RoboDK station: kr30 cnc 041619 kinda works.rdk

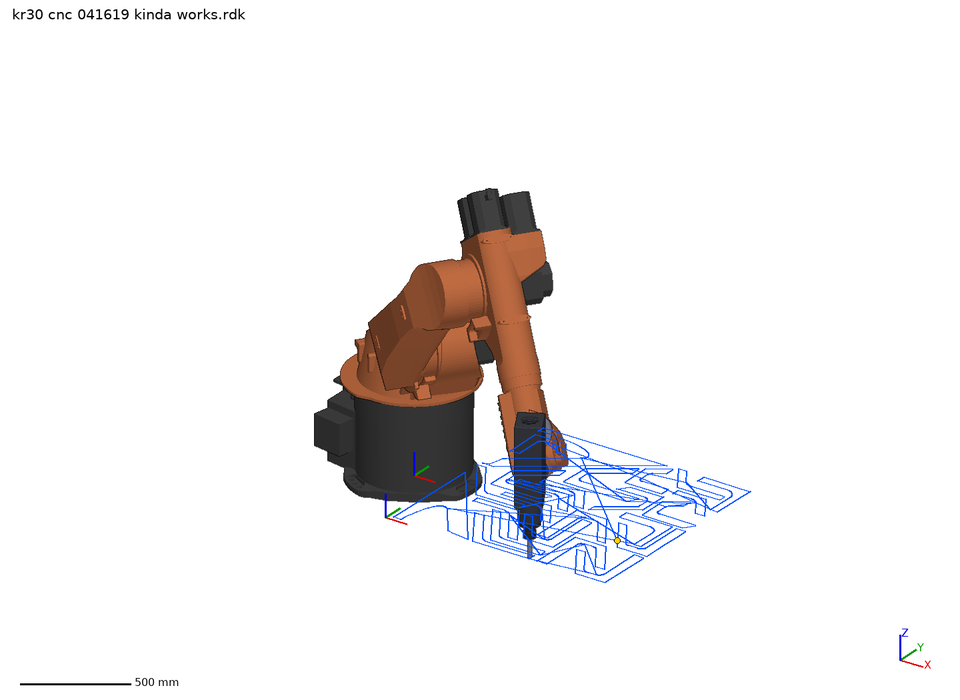
[picture v0: the station drawn from its stored meshes, robots at their saved joint values, targets as dots, program paths as lines]
Station kr30 cnc 041619 kinda works. Poses are relative to the parent item; angles as X-Y-Z fixed-axis rotations.
  - frame KUKA KR 30 HA Base at (0, 0, 0) mm
    - robot KUKA KR 30 HA: 6 axes, payload 30 kg, reach 2033 mm, repeatability 0.05 mm, weight 665 kg
        modified DH rows (alpha deg, a mm, theta deg, d mm): 0, 0, 0, 815; -90, 350, 0, 0; 0, 850, -90, 0; -90, 145, 0, 820; 90, 0, 0, 0; -90, 0, 180, 170
        joint limits [-185, -135, -120, -350, -119, -350] to [185, 35, 158, 350, 119, 350]; home [0, -90, 90, 0, 0, 0]; saved at [34.087, -43.037, 98.882, -30.893, -59.792, 16.754]
      - tool 1/2" End Mill TCP, TCP at (337.71, -2.2, 160.57) mm, size 692.9 x 170 x 256 mm
    - frame Reference Rhino at (671.61, -1183.62, 450.23) mm
      - object RhinoPart at (0, 0, 0) mm
  - machining project RhinoPart Settings: C:/Users/Julian Ramirez.DESKTOP-JVDE542/Desktop/ELMER SHEET 1 TEST 3.nc | rotZ(0) | rotX(0)*rotY(0) | rotZ(0)*rotY(270)
  - object box at (500, 500, 500) mm, size 250 x 250 x 250 mm, geometry from box.sld
  - program RhinoPart (703 instructions, listed below)
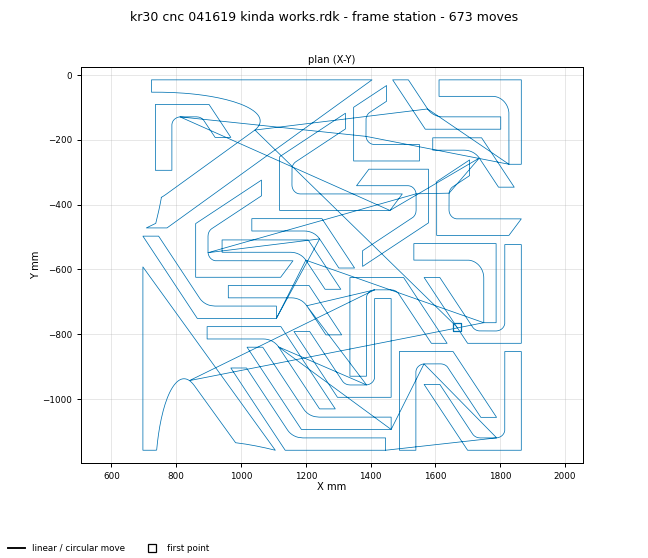
[picture p0: tool path of kr30 cnc 041619 kinda works.rdk in frame station, 673 of 673 moves have a stored position in this frame; points joined in program order, loops and branches not executed]

--- program RhinoPart (robot KUKA KR 30 HA) ---
  Smooth(1)
  Set Ref.: Reference Rhino
  Set Tool: 1/2" End Mill TCP
  Show 1/2" End Mill TCP
  Set speed (2000.0 mm/s)
  MoveJ 1 to (994.45, 406.4, 0) mm, rotated rx 0 ry 90 rz -60.43 deg; joints [17.989, -41.108, 95.853, -48.234, -64.788, 25.501]
  MoveL 2 to (994.45, 406.4, 0) mm, rotated rx 0 ry 90 rz -60.43 deg; joints [17.989, -41.108, 95.853, -48.234, -64.788, 25.501]
  MoveL 3 to (994.45, 406.4, 0) mm, rotated rx 0 ry 90 rz -60.43 deg; joints [17.989, -41.108, 95.853, -48.234, -64.788, 25.501]
  Set speed (60.0 mm/s)
  MoveL 4 to (1028.02, 355.6, 0) mm, rotated rx 0 ry 90 rz -60.43 deg; joints [19.323, -38.739, 90.931, -47.84, -62.49, 27.027]
  MoveL 5 to (1069.46, 355.6, 0) mm, rotated rx 0 ry 90 rz -60.43 deg; joints [18.852, -36.71, 86.73, -49.181, -61.272, 29.094]
  MoveL 6 to (1110.91, 355.6, 0) mm, rotated rx 0 ry 90 rz -60.43 deg; joints [18.403, -34.571, 82.311, -50.606, -60.029, 31.313]
  MoveL 7 to (1152.36, 355.6, 0) mm, rotated rx 0 ry 90 rz -60.43 deg; joints [17.974, -32.3, 77.632, -52.139, -58.757, 33.711]
  MoveL 8 to (1193.8, 355.6, 0) mm, rotated rx 0 ry 90 rz -60.43 deg; joints [17.564, -29.869, 72.637, -53.809, -57.448, 36.332]
  MoveL 9 to (1193.8, 431.8, 0) mm, rotated rx 0 ry 90 rz -60.43 deg; joints [15.206, -31.214, 75.401, -55.332, -59.663, 36.14]
  MoveL 10 to (1193.8, 508, 0) mm, rotated rx 0 ry 90 rz -60.43 deg; joints [12.795, -32.328, 77.69, -57.017, -61.74, 36.113]
  MoveL 11 to (1193.8, 584.2, 0) mm, rotated rx 0 ry 90 rz -60.43 deg; joints [10.336, -33.225, 79.537, -58.835, -63.695, 36.231]
  MoveL 12 to (1193.8, 660.4, 0) mm, rotated rx 0 ry 90 rz -60.43 deg; joints [7.839, -33.917, 80.962, -60.76, -65.545, 36.484]
  MoveL 13 to (1142.85, 660.4, 0) mm, rotated rx 0 ry 90 rz -60.43 deg; joints [8.077, -36.69, 86.686, -59.419, -66.88, 33.602]
  MoveL 14 to (1142.85, 419.1, 0) mm, rotated rx 0 ry 90 rz -60.43 deg; joints [16.06, -33.91, 80.949, -53.199, -60.845, 33.072]
  MoveL 15 to (1142.7, 416.47, 0) mm, rotated rx 0 ry 90 rz -60.43 deg; joints [16.145, -33.877, 80.88, -53.133, -60.777, 33.065]
  MoveL 16 to (1142.26, 413.91, 0) mm, rotated rx 0 ry 90 rz -60.43 deg; joints [16.231, -33.86, 80.846, -53.058, -60.719, 33.041]
  MoveL 17 to (1141.56, 411.43, 0) mm, rotated rx 0 ry 90 rz -60.43 deg; joints [16.317, -33.859, 80.844, -52.976, -60.672, 33.001]
  MoveL 18 to (1140.59, 409.05, 0) mm, rotated rx 0 ry 90 rz -60.43 deg; joints [16.402, -33.874, 80.874, -52.887, -60.635, 32.947]
  MoveL 19 to (1139.37, 406.78, 0) mm, rotated rx 0 ry 90 rz -60.43 deg; joints [16.486, -33.904, 80.935, -52.792, -60.609, 32.878]
  MoveL 20 to (1137.93, 404.64, 0) mm, rotated rx 0 ry 90 rz -60.43 deg; joints [16.568, -33.948, 81.027, -52.692, -60.593, 32.796]
  MoveL 21 to (1136.26, 402.65, 0) mm, rotated rx 0 ry 90 rz -60.43 deg; joints [16.648, -34.006, 81.147, -52.587, -60.587, 32.702]
  MoveL 22 to (1134.38, 400.81, 0) mm, rotated rx 0 ry 90 rz -60.43 deg; joints [16.724, -34.079, 81.296, -52.479, -60.592, 32.596]
  MoveL 23 to (1132.33, 399.17, 0) mm, rotated rx 0 ry 90 rz -60.43 deg; joints [16.796, -34.163, 81.47, -52.369, -60.608, 32.48]
  MoveL 24 to (1130.15, 397.73, 0) mm, rotated rx 0 ry 90 rz -60.43 deg; joints [16.863, -34.258, 81.665, -52.26, -60.634, 32.357]
  MoveL 25 to (1127.84, 396.51, 0) mm, rotated rx 0 ry 90 rz -60.43 deg; joints [16.925, -34.362, 81.88, -52.151, -60.669, 32.227]
  MoveL 26 to (1125.43, 395.51, 0) mm, rotated rx 0 ry 90 rz -60.43 deg; joints [16.981, -34.475, 82.113, -52.044, -60.713, 32.092]
  MoveL 27 to (1122.95, 394.72, 0) mm, rotated rx 0 ry 90 rz -60.43 deg; joints [17.03, -34.595, 82.361, -51.939, -60.765, 31.953]
  MoveL 28 to (1120.4, 394.16, 0) mm, rotated rx 0 ry 90 rz -60.43 deg; joints [17.073, -34.722, 82.623, -51.838, -60.826, 31.811]
  MoveL 29 to (1117.81, 393.81, 0) mm, rotated rx 0 ry 90 rz -60.43 deg; joints [17.11, -34.855, 82.896, -51.74, -60.893, 31.667]
  MoveL 30 to (1115.19, 393.7, 0) mm, rotated rx 0 ry 90 rz -60.43 deg; joints [17.14, -34.991, 83.179, -51.648, -60.968, 31.523]
  MoveL 31 to (1066.94, 393.7, 0) mm, rotated rx 0 ry 90 rz -60.43 deg; joints [17.632, -37.464, 88.289, -50.062, -62.386, 28.97]
  MoveL 32 to (1063.47, 393.9, 0) mm, rotated rx 0 ry 90 rz -60.43 deg; joints [17.662, -37.639, 88.651, -49.958, -62.492, 28.794]
  MoveL 33 to (1060.06, 394.5, 0) mm, rotated rx 0 ry 90 rz -60.43 deg; joints [17.678, -37.817, 89.019, -49.866, -62.606, 28.623]
  MoveL 34 to (1056.75, 395.49, 0) mm, rotated rx 0 ry 90 rz -60.43 deg; joints [17.68, -37.995, 89.388, -49.788, -62.728, 28.457]
  MoveL 35 to (1053.59, 396.85, 0) mm, rotated rx 0 ry 90 rz -60.43 deg; joints [17.668, -38.171, 89.753, -49.726, -62.856, 28.301]
  MoveL 36 to (1050.62, 398.59, 0) mm, rotated rx 0 ry 90 rz -60.43 deg; joints [17.642, -38.343, 90.109, -49.68, -62.988, 28.155]
  MoveL 37 to (1047.88, 400.69, 0) mm, rotated rx 0 ry 90 rz -60.43 deg; joints [17.601, -38.508, 90.452, -49.652, -63.122, 28.021]
  MoveL 38 to (1045.42, 403.13, 0) mm, rotated rx 0 ry 90 rz -60.43 deg; joints [17.545, -38.664, 90.776, -49.643, -63.257, 27.903]
  MoveL 39 to (1043.29, 405.92, 0) mm, rotated rx 0 ry 90 rz -60.43 deg; joints [17.474, -38.81, 91.077, -49.653, -63.391, 27.801]
  MoveL 40 to (942.25, 558.8, 0) mm, rotated rx 0 ry 90 rz -60.43 deg; joints [13.032, -45.298, 104.615, -51.659, -69.793, 23.593]
  MoveL 41 to (893.72, 558.8, 0) mm, rotated rx 0 ry 90 rz -60.43 deg; joints [13.466, -47.341, 108.919, -50.607, -71.044, 21.582]
  MoveL 42 to (927.3, 508, 0) mm, rotated rx 0 ry 90 rz -60.43 deg; joints [15.067, -45.394, 104.817, -49.631, -69.058, 22.803]
  MoveL 43 to (960.87, 457.2, 0) mm, rotated rx 0 ry 90 rz -60.43 deg; joints [16.572, -43.32, 100.47, -48.836, -66.974, 24.102]
  MoveL 44 to (994.45, 406.4, 0) mm, rotated rx 0 ry 90 rz -60.43 deg; joints [17.989, -41.108, 95.853, -48.234, -64.788, 25.501]
  MoveL 45 to (371.32, 1014.09, 0) mm, rotated rx 0 ry 90 rz -60.43 deg; joints [-7.691, -66.672, 152.583, -68.17, -88.477, 3.796]
  Set speed (60.0 mm/s)
  MoveL 46 to (375.76, 1018.13, 0) mm, rotated rx 0 ry 90 rz -60.43 deg; joints [-7.909, -66.538, 152.227, -68.394, -88.41, 4.007]
  MoveL 47 to (379.48, 1022.21, 0) mm, rotated rx 0 ry 90 rz -60.43 deg; joints [-8.134, -66.421, 151.921, -68.623, -88.357, 4.19]
  MoveL 48 to (382.49, 1026.31, 0) mm, rotated rx 0 ry 90 rz -60.43 deg; joints [-8.365, -66.323, 151.664, -68.857, -88.316, 4.345]
  MoveL 49 to (384.79, 1030.42, 0) mm, rotated rx 0 ry 90 rz -60.43 deg; joints [-8.601, -66.244, 151.456, -69.096, -88.288, 4.472]
  MoveL 50 to (386.4, 1034.54, 0) mm, rotated rx 0 ry 90 rz -60.43 deg; joints [-8.843, -66.182, 151.296, -69.341, -88.272, 4.571]
  MoveL 51 to (387.31, 1038.67, 0) mm, rotated rx 0 ry 90 rz -60.43 deg; joints [-9.091, -66.14, 151.185, -69.59, -88.268, 4.643]
  MoveL 52 to (387.53, 1042.79, 0) mm, rotated rx 0 ry 90 rz -60.43 deg; joints [-9.345, -66.115, 151.121, -69.844, -88.275, 4.687]
  MoveL 53 to (387.07, 1046.9, 0) mm, rotated rx 0 ry 90 rz -60.43 deg; joints [-9.606, -66.109, 151.105, -70.104, -88.293, 4.704]
  MoveL 54 to (385.93, 1051, 0) mm, rotated rx 0 ry 90 rz -60.43 deg; joints [-9.872, -66.121, 151.137, -70.369, -88.322, 4.694]
  MoveL 55 to (384.11, 1055.07, 0) mm, rotated rx 0 ry 90 rz -60.43 deg; joints [-10.144, -66.151, 151.215, -70.639, -88.36, 4.657]
  MoveL 56 to (381.63, 1059.1, 0) mm, rotated rx 0 ry 90 rz -60.43 deg; joints [-10.423, -66.199, 151.339, -70.915, -88.408, 4.592]
  MoveL 57 to (378.49, 1063.11, 0) mm, rotated rx 0 ry 90 rz -60.43 deg; joints [-10.708, -66.264, 151.509, -71.197, -88.464, 4.501]
  MoveL 58 to (374.68, 1067.06, 0) mm, rotated rx 0 ry 90 rz -60.43 deg; joints [-11, -66.346, 151.724, -71.485, -88.529, 4.382]
  MoveL 59 to (370.23, 1070.97, 0) mm, rotated rx 0 ry 90 rz -60.43 deg; joints [-11.299, -66.446, 151.984, -71.779, -88.603, 4.237]
  MoveL 60 to (365.13, 1074.81, 0) mm, rotated rx 0 ry 90 rz -60.43 deg; joints [-11.605, -66.561, 152.289, -72.08, -88.683, 4.064]
  MoveL 61 to (356.11, 1080.56, 0) mm, rotated rx 0 ry 90 rz -60.43 deg; joints [-12.086, -66.768, 152.839, -72.553, -88.82, 3.748]
  MoveL 62 to (346.45, 1085.73, 0) mm, rotated rx 0 ry 90 rz -60.43 deg; joints [-12.548, -66.991, 153.437, -73.007, -88.96, 3.399]
  MoveL 63 to (336.49, 1090.32, 0) mm, rotated rx 0 ry 90 rz -60.43 deg; joints [-12.986, -67.22, 154.06, -73.438, -89.098, 3.029]
  MoveL 64 to (326.6, 1094.34, 0) mm, rotated rx 0 ry 90 rz -60.43 deg; joints [-13.395, -67.447, 154.682, -73.841, -89.23, 2.655]
  MoveL 65 to (304.84, 1101.8, 0) mm, rotated rx 0 ry 90 rz -60.43 deg; joints [-14.233, -67.937, 156.062, -74.669, -89.504, 1.809]
  MoveL 66 to (282.07, 1108.12, 0) mm, rotated rx 0 ry 90 rz -60.43 deg; joints [-15.052, -68.435, 157.512, -75.482, -89.769, 0.893]
  MoveL 67 to (259.04, 1113.38, 0) mm, rotated rx -90 ry 80 rz -150.43 deg; joints [-16.774, -66.906, 154.911, -77.21, -89.558, 11.945]
  MoveL 68 to (236.49, 1117.66, 0) mm, rotated rx -90 ry 80 rz -150.43 deg; joints [-17.5, -67.391, 156.356, -77.931, -89.784, 11.012]
  MoveL 69 to (215.72, 1120.95, 0) mm, rotated rx -90 ry 80 rz -150.43 deg; joints [-18.157, -67.818, 157.686, -78.586, -89.974, 10.13]
  MoveL 70 to (194.75, 1123.72, 0) mm, rotated rx -90 ry 70 rz -150.43 deg; joints [-19.526, -65.161, 154.981, -79.954, -89.969, 20.176]
  MoveL 71 to (173.72, 1126.01, 0) mm, rotated rx -90 ry 70 rz -150.43 deg; joints [-20.155, -65.544, 156.331, -80.584, -90.129, 19.224]
  MoveL 72 to (152.78, 1127.82, 0) mm, rotated rx -90 ry 70 rz -150.43 deg; joints [-20.781, -65.901, 157.673, -81.213, -90.271, 18.248]
  MoveL 73 to (132.99, 1129.14, 0) mm, rotated rx -90 ry 60 rz -150.43 deg; joints [-21.884, -62.292, 155, -82.321, -90.362, 27.317]
  MoveL 74 to (116.9, 1129.95, 0) mm, rotated rx -90 ry 60 rz -150.43 deg; joints [-22.346, -62.501, 156.03, -82.788, -90.444, 26.499]
  MoveL 75 to (100.77, 1130.52, 0) mm, rotated rx -90 ry 60 rz -150.43 deg; joints [-22.81, -62.691, 157.062, -83.258, -90.514, 25.659]
  MoveL 76 to (84.64, 1130.87, 0) mm, rotated rx -90 ry 50 rz -150.43 deg; joints [-23.629, -58.3, 154.305, -84.09, -90.621, 34.027]
  MoveL 77 to (68.52, 1130.98, 0) mm, rotated rx -90 ry 50 rz -150.43 deg; joints [-24.076, -58.406, 155.332, -84.545, -90.662, 33.106]
  MoveL 78 to (51.93, 1130.98, 0) mm, rotated rx -90 ry 50 rz -150.43 deg; joints [-24.547, -58.489, 156.384, -85.022, -90.689, 32.135]
  MoveL 79 to (51.93, 1169.08, 0) mm, rotated rx -90 ry 50 rz -150.43 deg; joints [-26.906, -58.397, 155.233, -87.353, -90.317, 33.172]
  MoveL 80 to (732.85, 1169.08, 0) mm, rotated rx 0 ry 90 rz -60.43 deg; joints [-12.432, -54.145, 123.468, -73.905, -84.027, 19.832]
  MoveL 81 to (99.83, 711.88, 0) mm, rotated rx -90 ry 50 rz -150.43 deg; joints [5.455, -58.558, 157.979, -55.338, -95.391, 32.262]
  MoveL 82 to (36.02, 711.88, 0) mm, rotated rx -90 ry 30 rz -150.43 deg; joints [2.816, -47.382, 156.026, -58.993, -99.86, 44.097]
  MoveL 83 to (65.11, 725.98, 0) mm, rotated rx -90 ry 40 rz -150.43 deg; joints [2.988, -53.284, 157.255, -58.216, -97.466, 38.157]
  MoveL 84 to (69.92, 745.6, 0) mm, rotated rx -90 ry 40 rz -150.43 deg; joints [1.576, -53.317, 156.983, -59.576, -97.019, 38.245]
  MoveL 85 to (74.45, 765.38, 0) mm, rotated rx -90 ry 40 rz -150.43 deg; joints [0.167, -53.349, 156.698, -60.933, -96.576, 38.358]
  MoveL 86 to (78.62, 785.23, 0) mm, rotated rx -90 ry 40 rz -150.43 deg; joints [-1.232, -53.378, 156.403, -62.28, -96.141, 38.492]
  MoveL 87 to (82.38, 805.12, 0) mm, rotated rx -90 ry 40 rz -150.43 deg; joints [-2.62, -53.405, 156.103, -63.617, -95.718, 38.643]
  MoveL 88 to (81.84, 806.04, 0) mm, rotated rx -90 ry 40 rz -150.43 deg; joints [-2.686, -53.402, 156.137, -63.686, -95.721, 38.604]
  MoveL 89 to (85.5, 808.13, 0) mm, rotated rx -90 ry 40 rz -150.43 deg; joints [-2.82, -53.422, 155.882, -63.793, -95.573, 38.839]
  MoveL 90 to (89.1, 810.32, 0) mm, rotated rx -90 ry 40 rz -150.43 deg; joints [-2.959, -53.44, 155.63, -63.907, -95.427, 39.069]
  MoveL 91 to (92.62, 812.61, 0) mm, rotated rx -90 ry 40 rz -150.43 deg; joints [-3.104, -53.455, 155.382, -64.028, -95.285, 39.293]
  MoveL 92 to (96.07, 815.01, 0) mm, rotated rx -90 ry 40 rz -150.43 deg; joints [-3.257, -53.469, 155.138, -64.158, -95.144, 39.512]
  MoveL 93 to (366.16, 1010.08, 0) mm, rotated rx 0 ry 90 rz -60.43 deg; joints [-7.478, -66.824, 152.988, -67.951, -88.558, 3.555]
  MoveL 94 to (371.32, 1014.09, 0) mm, rotated rx 0 ry 90 rz -60.43 deg; joints [-7.691, -66.672, 152.583, -68.17, -88.477, 3.796]
  MoveL 95 to (904.53, 1079.22, 0) mm, rotated rx 0 ry 90 rz -60.43 deg; joints [-7.417, -48.055, 110.429, -70.163, -79.93, 25.861]
  Set speed (60.0 mm/s)
  MoveL 96 to (845.14, 1169.08, 0) mm, rotated rx 0 ry 90 rz -60.43 deg; joints [-11.43, -49.863, 114.267, -73.538, -82.269, 24.476]
  MoveL 97 to (796.61, 1169.08, 0) mm, rotated rx 0 ry 90 rz -60.43 deg; joints [-11.843, -51.756, 118.313, -73.653, -83.042, 22.442]
  MoveL 98 to (897.33, 1016.68, 0) mm, rotated rx 0 ry 90 rz -60.43 deg; joints [-4.939, -48.634, 111.655, -67.774, -79.101, 24.832]
  MoveL 99 to (1130.3, 1016.68, 0) mm, rotated rx 0 ry 90 rz -60.43 deg; joints [-4.241, -37.976, 89.349, -69.706, -74.509, 35.838]
  MoveL 100 to (1130.3, 1054.78, 0) mm, rotated rx 0 ry 90 rz -60.43 deg; joints [-5.562, -37.808, 89.001, -70.857, -75.226, 36.302]
  MoveL 101 to (951.82, 1054.78, 0) mm, rotated rx 0 ry 90 rz -60.43 deg; joints [-6.235, -46.179, 106.468, -69.459, -78.678, 27.653]
  MoveL 102 to (948.36, 1054.88, 0) mm, rotated rx 0 ry 90 rz -60.43 deg; joints [-6.254, -46.327, 106.78, -69.445, -78.744, 27.499]
  MoveL 103 to (944.91, 1055.18, 0) mm, rotated rx 0 ry 90 rz -60.43 deg; joints [-6.28, -46.474, 107.089, -69.439, -78.813, 27.349]
  MoveL 104 to (941.49, 1055.67, 0) mm, rotated rx 0 ry 90 rz -60.43 deg; joints [-6.314, -46.618, 107.393, -69.44, -78.884, 27.203]
  MoveL 105 to (938.11, 1056.36, 0) mm, rotated rx 0 ry 90 rz -60.43 deg; joints [-6.356, -46.759, 107.69, -69.449, -78.958, 27.061]
  MoveL 106 to (934.77, 1057.25, 0) mm, rotated rx 0 ry 90 rz -60.43 deg; joints [-6.405, -46.897, 107.981, -69.466, -79.034, 26.923]
  MoveL 107 to (931.49, 1058.34, 0) mm, rotated rx 0 ry 90 rz -60.43 deg; joints [-6.462, -47.031, 108.264, -69.491, -79.112, 26.791]
  MoveL 108 to (928.27, 1059.61, 0) mm, rotated rx 0 ry 90 rz -60.43 deg; joints [-6.527, -47.161, 108.539, -69.524, -79.192, 26.664]
  MoveL 109 to (925.13, 1061.08, 0) mm, rotated rx 0 ry 90 rz -60.43 deg; joints [-6.599, -47.286, 108.803, -69.564, -79.273, 26.544]
  MoveL 110 to (922.08, 1062.74, 0) mm, rotated rx 0 ry 90 rz -60.43 deg; joints [-6.678, -47.407, 109.058, -69.613, -79.355, 26.429]
  MoveL 111 to (919.14, 1064.59, 0) mm, rotated rx 0 ry 90 rz -60.43 deg; joints [-6.765, -47.521, 109.3, -69.67, -79.438, 26.322]
  MoveL 112 to (916.32, 1066.61, 0) mm, rotated rx 0 ry 90 rz -60.43 deg; joints [-6.858, -47.629, 109.528, -69.734, -79.521, 26.223]
  MoveL 113 to (913.65, 1068.81, 0) mm, rotated rx 0 ry 90 rz -60.43 deg; joints [-6.958, -47.73, 109.741, -69.805, -79.604, 26.132]
  MoveL 114 to (911.12, 1071.17, 0) mm, rotated rx 0 ry 90 rz -60.43 deg; joints [-7.064, -47.824, 109.939, -69.884, -79.687, 26.05]
  MoveL 115 to (908.75, 1073.7, 0) mm, rotated rx 0 ry 90 rz -60.43 deg; joints [-7.176, -47.909, 110.12, -69.971, -79.769, 25.977]
  MoveL 116 to (906.55, 1076.38, 0) mm, rotated rx 0 ry 90 rz -60.43 deg; joints [-7.294, -47.987, 110.284, -70.064, -79.85, 25.914]
  MoveL 117 to (904.53, 1079.22, 0) mm, rotated rx 0 ry 90 rz -60.43 deg; joints [-7.417, -48.055, 110.429, -70.163, -79.93, 25.861]
  MoveL 118 to (1155.7, 908.41, 0) mm, rotated rx 0 ry 90 rz -60.43 deg; joints [-0.46, -36.883, 87.087, -66.837, -71.857, 36.048]
  Set speed (60.0 mm/s)
  MoveL 119 to (1155.7, 1062.81, 0) mm, rotated rx 0 ry 90 rz -60.43 deg; joints [-5.751, -36.438, 86.167, -71.384, -74.866, 37.777]
  MoveL 120 to (1155.47, 1068.04, 0) mm, rotated rx 0 ry 90 rz -60.43 deg; joints [-5.93, -36.422, 86.133, -71.535, -74.971, 37.832]
  MoveL 121 to (1154.79, 1073.23, 0) mm, rotated rx 0 ry 90 rz -60.43 deg; joints [-6.109, -36.429, 86.148, -71.679, -75.083, 37.862]
  MoveL 122 to (1153.66, 1078.33, 0) mm, rotated rx 0 ry 90 rz -60.43 deg; joints [-6.286, -36.46, 86.211, -71.816, -75.202, 37.867]
  MoveL 123 to (1152.09, 1083.3, 0) mm, rotated rx 0 ry 90 rz -60.43 deg; joints [-6.461, -36.514, 86.323, -71.945, -75.327, 37.847]
  MoveL 124 to (1150.07, 1088.11, 0) mm, rotated rx 0 ry 90 rz -60.43 deg; joints [-6.633, -36.591, 86.483, -72.064, -75.458, 37.802]
  MoveL 125 to (1147.63, 1092.73, 0) mm, rotated rx 0 ry 90 rz -60.43 deg; joints [-6.8, -36.691, 86.69, -72.174, -75.593, 37.73]
  MoveL 126 to (1144.76, 1097.1, 0) mm, rotated rx 0 ry 90 rz -60.43 deg; joints [-6.961, -36.815, 86.945, -72.274, -75.732, 37.633]
  MoveL 127 to (1141.47, 1101.2, 0) mm, rotated rx 0 ry 90 rz -60.43 deg; joints [-7.115, -36.961, 87.247, -72.362, -75.873, 37.511]
  MoveL 128 to (1137.81, 1104.95, 0) mm, rotated rx 0 ry 90 rz -60.43 deg; joints [-7.259, -37.127, 87.592, -72.437, -76.014, 37.364]
  MoveL 129 to (1133.82, 1108.29, 0) mm, rotated rx 0 ry 90 rz -60.43 deg; joints [-7.39, -37.312, 87.975, -72.498, -76.154, 37.196]
  MoveL 130 to (1129.54, 1111.18, 0) mm, rotated rx 0 ry 90 rz -60.43 deg; joints [-7.509, -37.514, 88.393, -72.545, -76.29, 37.007]
  MoveL 131 to (1125, 1113.61, 0) mm, rotated rx 0 ry 90 rz -60.43 deg; joints [-7.613, -37.731, 88.842, -72.577, -76.422, 36.799]
  MoveL 132 to (1120.24, 1115.55, 0) mm, rotated rx 0 ry 90 rz -60.43 deg; joints [-7.702, -37.962, 89.32, -72.594, -76.549, 36.574]
  MoveL 133 to (1115.28, 1116.96, 0) mm, rotated rx 0 ry 90 rz -60.43 deg; joints [-7.774, -38.204, 89.823, -72.594, -76.67, 36.332]
  MoveL 134 to (1110.15, 1117.83, 0) mm, rotated rx 0 ry 90 rz -60.43 deg; joints [-7.829, -38.458, 90.347, -72.578, -76.784, 36.077]
  MoveL 135 to (1104.9, 1118.13, 0) mm, rotated rx 0 ry 90 rz -60.43 deg; joints [-7.864, -38.72, 90.891, -72.545, -76.889, 35.807]
  MoveL 136 to (939.8, 1118.13, 0) mm, rotated rx 0 ry 90 rz -60.43 deg; joints [-8.746, -46.337, 106.801, -71.688, -79.906, 27.905]
  MoveL 137 to (939.8, 1169.08, 0) mm, rotated rx 0 ry 90 rz -60.43 deg; joints [-10.702, -45.963, 106.015, -73.503, -80.708, 28.599]
  MoveL 138 to (1193.8, 1169.08, 0) mm, rotated rx 0 ry 90 rz -60.43 deg; joints [-9.136, -33.584, 80.276, -74.83, -76.143, 41.453]
  MoveL 139 to (1193.8, 908.41, 0) mm, rotated rx 0 ry 90 rz -60.43 deg; joints [-0.45, -34.818, 82.821, -67.51, -70.997, 38.185]
  MoveL 140 to (1155.7, 908.41, 0) mm, rotated rx 0 ry 90 rz -60.43 deg; joints [-0.46, -36.883, 87.087, -66.837, -71.857, 36.048]
  MoveL 141 to (714.35, 994.58, 0) mm, rotated rx 0 ry 90 rz -60.43 deg; joints [-4.647, -55.782, 127.04, -66.248, -82.218, 17.103]
  Set speed (60.0 mm/s)
  MoveL 142 to (714.24, 997.2, 0) mm, rotated rx 0 ry 90 rz -60.43 deg; joints [-4.769, -55.778, 127.032, -66.366, -82.252, 17.123]
  MoveL 143 to (714.24, 1045.45, 0) mm, rotated rx 0 ry 90 rz -60.43 deg; joints [-7.003, -55.598, 126.636, -68.542, -82.836, 17.603]
  MoveL 144 to (714.44, 1048.91, 0) mm, rotated rx 0 ry 90 rz -60.43 deg; joints [-7.161, -55.575, 126.586, -68.697, -82.874, 17.647]
  MoveL 145 to (715.04, 1052.32, 0) mm, rotated rx 0 ry 90 rz -60.43 deg; joints [-7.315, -55.537, 126.504, -68.85, -82.905, 17.707]
  MoveL 146 to (716.03, 1055.63, 0) mm, rotated rx 0 ry 90 rz -60.43 deg; joints [-7.461, -55.486, 126.391, -68.997, -82.927, 17.782]
  MoveL 147 to (717.39, 1058.8, 0) mm, rotated rx 0 ry 90 rz -60.43 deg; joints [-7.598, -55.421, 126.25, -69.138, -82.942, 17.871]
  MoveL 148 to (719.13, 1061.77, 0) mm, rotated rx 0 ry 90 rz -60.43 deg; joints [-7.723, -55.344, 126.08, -69.268, -82.948, 17.972]
  MoveL 149 to (721.23, 1064.5, 0) mm, rotated rx 0 ry 90 rz -60.43 deg; joints [-7.835, -55.254, 125.883, -69.388, -82.945, 18.086]
  MoveL 150 to (723.67, 1066.96, 0) mm, rotated rx 0 ry 90 rz -60.43 deg; joints [-7.932, -55.152, 125.661, -69.494, -82.932, 18.211]
  MoveL 151 to (726.46, 1069.09, 0) mm, rotated rx 0 ry 90 rz -60.43 deg; joints [-8.011, -55.039, 125.415, -69.586, -82.911, 18.346]
  MoveL 152 to (777.74, 1102.98, 0) mm, rotated rx 0 ry 90 rz -60.43 deg; joints [-9.171, -52.942, 120.865, -70.984, -82.472, 20.814]
  MoveL 153 to (777.74, 1151.51, 0) mm, rotated rx 0 ry 90 rz -60.43 deg; joints [-11.262, -52.611, 120.151, -72.996, -83.107, 21.428]
  MoveL 154 to (676.14, 1084.36, 0) mm, rotated rx 0 ry 90 rz -60.43 deg; joints [-9.067, -56.765, 129.203, -70.376, -83.933, 16.512]
  MoveL 155 to (676.14, 918.58, 0) mm, rotated rx 0 ry 90 rz -60.43 deg; joints [-1.138, -57.291, 130.366, -62.615, -82.032, 14.981]
  MoveL 156 to (879.34, 918.58, 0) mm, rotated rx 0 ry 90 rz -60.43 deg; joints [-0.971, -49.58, 113.665, -63.877, -77.924, 23.104]
  MoveL 157 to (879.34, 969.54, 0) mm, rotated rx 0 ry 90 rz -60.43 deg; joints [-3.069, -49.507, 113.509, -65.859, -78.72, 23.578]
  MoveL 158 to (739.64, 969.54, 0) mm, rotated rx 0 ry 90 rz -60.43 deg; joints [-3.412, -54.921, 125.157, -65.191, -81.426, 17.875]
  MoveL 159 to (737.01, 969.69, 0) mm, rotated rx 0 ry 90 rz -60.43 deg; joints [-3.425, -55.017, 125.367, -65.189, -81.478, 17.772]
  MoveL 160 to (734.45, 970.12, 0) mm, rotated rx 0 ry 90 rz -60.43 deg; joints [-3.452, -55.111, 125.571, -65.2, -81.533, 17.675]
  MoveL 161 to (731.97, 970.83, 0) mm, rotated rx 0 ry 90 rz -60.43 deg; joints [-3.492, -55.2, 125.767, -65.223, -81.589, 17.583]
  MoveL 162 to (729.59, 971.8, 0) mm, rotated rx 0 ry 90 rz -60.43 deg; joints [-3.543, -55.286, 125.953, -65.259, -81.647, 17.497]
  MoveL 163 to (727.32, 973.01, 0) mm, rotated rx 0 ry 90 rz -60.43 deg; joints [-3.605, -55.366, 126.129, -65.307, -81.706, 17.419]
  MoveL 164 to (725.18, 974.46, 0) mm, rotated rx 0 ry 90 rz -60.43 deg; joints [-3.679, -55.441, 126.293, -65.365, -81.765, 17.347]
  MoveL 165 to (723.19, 976.13, 0) mm, rotated rx 0 ry 90 rz -60.43 deg; joints [-3.762, -55.51, 126.444, -65.435, -81.823, 17.283]
  MoveL 166 to (721.35, 978, 0) mm, rotated rx 0 ry 90 rz -60.43 deg; joints [-3.854, -55.572, 126.58, -65.514, -81.882, 17.228]
  MoveL 167 to (719.71, 980.05, 0) mm, rotated rx 0 ry 90 rz -60.43 deg; joints [-3.954, -55.627, 126.7, -65.603, -81.938, 17.181]
  MoveL 168 to (718.27, 982.24, 0) mm, rotated rx 0 ry 90 rz -60.43 deg; joints [-4.06, -55.674, 126.802, -65.698, -81.992, 17.145]
  MoveL 169 to (717.05, 984.54, 0) mm, rotated rx 0 ry 90 rz -60.43 deg; joints [-4.171, -55.712, 126.887, -65.799, -82.044, 17.117]
  MoveL 170 to (716.05, 986.95, 0) mm, rotated rx 0 ry 90 rz -60.43 deg; joints [-4.287, -55.742, 126.953, -65.906, -82.093, 17.1]
  MoveL 171 to (715.26, 989.44, 0) mm, rotated rx 0 ry 90 rz -60.43 deg; joints [-4.405, -55.764, 127, -66.017, -82.138, 17.091]
  MoveL 172 to (714.69, 991.99, 0) mm, rotated rx 0 ry 90 rz -60.43 deg; joints [-4.526, -55.777, 127.029, -66.131, -82.18, 17.093]
  MoveL 173 to (714.35, 994.58, 0) mm, rotated rx 0 ry 90 rz -60.43 deg; joints [-4.647, -55.782, 127.04, -66.248, -82.218, 17.103]
  MoveL 174 to (139.93, 1054.78, 0) mm, rotated rx -90 ry 60 rz -150.43 deg; joints [-16.954, -62.55, 156.283, -77.409, -90.815, 26.356]
  Set speed (60.0 mm/s)
  MoveL 175 to (137.34, 1054.44, 0) mm, rotated rx -90 ry 60 rz -150.43 deg; joints [-16.984, -62.584, 156.465, -77.44, -90.845, 26.212]
  MoveL 176 to (134.79, 1053.88, 0) mm, rotated rx -90 ry 60 rz -150.43 deg; joints [-16.998, -62.617, 156.648, -77.457, -90.877, 26.066]
  MoveL 177 to (132.3, 1053.09, 0) mm, rotated rx -90 ry 60 rz -150.43 deg; joints [-16.996, -62.65, 156.831, -77.457, -90.91, 25.919]
  MoveL 178 to (129.9, 1052.08, 0) mm, rotated rx -90 ry 60 rz -150.43 deg; joints [-16.978, -62.682, 157.013, -77.442, -90.943, 25.773]
  MoveL 179 to (127.59, 1050.86, 0) mm, rotated rx -90 ry 60 rz -150.43 deg; joints [-16.944, -62.714, 157.193, -77.41, -90.978, 25.628]
  MoveL 180 to (125.4, 1049.43, 0) mm, rotated rx -90 ry 60 rz -150.43 deg; joints [-16.892, -62.743, 157.37, -77.361, -91.014, 25.486]
  MoveL 181 to (123.35, 1047.78, 0) mm, rotated rx -90 ry 60 rz -150.43 deg; joints [-16.824, -62.772, 157.541, -77.295, -91.051, 25.348]
  MoveL 182 to (121.48, 1045.95, 0) mm, rotated rx -90 ry 60 rz -150.43 deg; joints [-16.738, -62.798, 157.704, -77.212, -91.088, 25.217]
  MoveL 183 to (119.81, 1043.95, 0) mm, rotated rx -90 ry 60 rz -150.43 deg; joints [-16.637, -62.822, 157.856, -77.114, -91.125, 25.094]
  MoveL 184 to (118.36, 1041.82, 0) mm, rotated rx -90 ry 60 rz -150.43 deg; joints [-16.521, -62.844, 157.995, -77.001, -91.162, 24.981]
  MoveL 185 to (117.15, 1039.55, 0) mm, rotated rx -90 ry 50 rz -150.43 deg; joints [-17.126, -58.31, 154.398, -77.622, -91.31, 34.054]
  MoveL 186 to (116.18, 1037.16, 0) mm, rotated rx -90 ry 50 rz -150.43 deg; joints [-16.992, -58.323, 154.512, -77.491, -91.345, 33.959]
  MoveL 187 to (115.47, 1034.68, 0) mm, rotated rx -90 ry 50 rz -150.43 deg; joints [-16.846, -58.334, 154.61, -77.348, -91.38, 33.877]
  MoveL 188 to (115.04, 1032.12, 0) mm, rotated rx -90 ry 50 rz -150.43 deg; joints [-16.689, -58.343, 154.69, -77.194, -91.412, 33.811]
  MoveL 189 to (114.89, 1029.5, 0) mm, rotated rx -90 ry 50 rz -150.43 deg; joints [-16.522, -58.349, 154.753, -77.029, -91.443, 33.761]
  MoveL 190 to (114.89, 889.8, 0) mm, rotated rx -90 ry 50 rz -150.43 deg; joints [-7.121, -58.512, 156.752, -67.759, -93.138, 32.377]
  MoveL 191 to (63.94, 889.8, 0) mm, rotated rx -90 ry 40 rz -150.43 deg; joints [-8.69, -53.34, 156.782, -69.643, -94.753, 37.412]
  MoveL 192 to (63.94, 1093, 0) mm, rotated rx -90 ry 50 rz -150.43 deg; joints [-21.787, -58.506, 156.655, -82.293, -91.1, 31.925]
  MoveL 193 to (229.71, 1093, 0) mm, rotated rx -90 ry 80 rz -150.43 deg; joints [-16.004, -67.703, 157.32, -76.433, -89.91, 10.372]
  MoveL 194 to (296.86, 991.4, 0) mm, rotated rx -90 ry 80 rz -150.43 deg; joints [-8.306, -66.648, 154.164, -68.753, -89.099, 12.315]
  MoveL 195 to (248.33, 991.4, 0) mm, rotated rx -90 ry 80 rz -150.43 deg; joints [-8.797, -67.784, 157.578, -69.225, -89.927, 10.193]
  MoveL 196 to (214.44, 1042.68, 0) mm, rotated rx -90 ry 70 rz -150.43 deg; joints [-13.925, -65.253, 155.3, -74.354, -90.013, 19.955]
  MoveL 197 to (212.31, 1045.46, 0) mm, rotated rx -90 ry 70 rz -150.43 deg; joints [-14.142, -65.281, 155.398, -74.571, -90.031, 19.887]
  MoveL 198 to (209.86, 1047.91, 0) mm, rotated rx -90 ry 70 rz -150.43 deg; joints [-14.343, -65.318, 155.525, -74.772, -90.054, 19.8]
  MoveL 199 to (207.12, 1050.01, 0) mm, rotated rx -90 ry 70 rz -150.43 deg; joints [-14.527, -65.361, 155.676, -74.956, -90.082, 19.696]
  MoveL 200 to (204.15, 1051.74, 0) mm, rotated rx -90 ry 70 rz -150.43 deg; joints [-14.692, -65.41, 155.849, -75.121, -90.113, 19.576]
  MoveL 201 to (200.98, 1053.11, 0) mm, rotated rx -90 ry 70 rz -150.43 deg; joints [-14.837, -65.463, 156.041, -75.266, -90.147, 19.441]
  MoveL 202 to (197.68, 1054.1, 0) mm, rotated rx -90 ry 70 rz -150.43 deg; joints [-14.96, -65.521, 156.25, -75.39, -90.184, 19.295]
  MoveL 203 to (190.8, 1054.9, 0) mm, rotated rx -90 ry 70 rz -150.43 deg; joints [-15.136, -65.646, 156.705, -75.567, -90.264, 18.974]
  MoveL 204 to (142.55, 1054.9, 0) mm, rotated rx -90 ry 60 rz -150.43 deg; joints [-16.91, -62.515, 156.104, -77.362, -90.786, 26.498]
  MoveL 205 to (139.93, 1054.78, 0) mm, rotated rx -90 ry 60 rz -150.43 deg; joints [-16.954, -62.55, 156.283, -77.409, -90.815, 26.356]
  MoveL 206 to (788.26, 765.88, 0) mm, rotated rx 0 ry 90 rz -60.43 deg; joints [5.679, -52.932, 120.844, -56.78, -77.465, 18.335]
  Set speed (60.0 mm/s)
  MoveL 207 to (826.36, 816.83, 0) mm, rotated rx 0 ry 90 rz -60.43 deg; joints [3.348, -51.614, 118.009, -59.322, -77.431, 20.144]
  MoveL 208 to (511.04, 816.83, 0) mm, rotated rx 0 ry 90 rz -60.43 deg; joints [4.378, -62.718, 142.747, -56.454, -84.451, 8.298]
  MoveL 209 to (505.85, 817.41, 0) mm, rotated rx 0 ry 90 rz -60.43 deg; joints [4.367, -62.881, 143.134, -56.446, -84.576, 8.111]
  MoveL 210 to (503.37, 818.12, 0) mm, rotated rx 0 ry 90 rz -60.43 deg; joints [4.338, -62.96, 143.321, -56.467, -84.64, 8.023]
  MoveL 211 to (500.99, 819.09, 0) mm, rotated rx 0 ry 90 rz -60.43 deg; joints [4.294, -63.036, 143.503, -56.502, -84.704, 7.939]
  MoveL 212 to (498.72, 820.3, 0) mm, rotated rx 0 ry 90 rz -60.43 deg; joints [4.235, -63.11, 143.677, -56.553, -84.768, 7.859]
  MoveL 213 to (496.58, 821.75, 0) mm, rotated rx 0 ry 90 rz -60.43 deg; joints [4.162, -63.179, 143.843, -56.619, -84.831, 7.785]
  MoveL 214 to (494.59, 823.42, 0) mm, rotated rx 0 ry 90 rz -60.43 deg; joints [4.075, -63.244, 143.999, -56.698, -84.893, 7.717]
  MoveL 215 to (492.75, 825.29, 0) mm, rotated rx 0 ry 90 rz -60.43 deg; joints [3.976, -63.305, 144.144, -56.79, -84.952, 7.655]
  MoveL 216 to (491.11, 827.34, 0) mm, rotated rx 0 ry 90 rz -60.43 deg; joints [3.866, -63.36, 144.276, -56.894, -85.009, 7.6]
  MoveL 217 to (489.67, 829.53, 0) mm, rotated rx 0 ry 90 rz -60.43 deg; joints [3.747, -63.408, 144.392, -57.008, -85.062, 7.553]
  MoveL 218 to (487.45, 834.24, 0) mm, rotated rx 0 ry 90 rz -60.43 deg; joints [3.486, -63.486, 144.578, -57.26, -85.155, 7.484]
  MoveL 219 to (486.09, 839.28, 0) mm, rotated rx 0 ry 90 rz -60.43 deg; joints [3.202, -63.536, 144.699, -57.537, -85.23, 7.447]
  MoveL 220 to (485.64, 844.49, 0) mm, rotated rx 0 ry 90 rz -60.43 deg; joints [2.904, -63.559, 144.753, -57.831, -85.285, 7.445]
  MoveL 221 to (485.64, 892.74, 0) mm, rotated rx 0 ry 90 rz -60.43 deg; joints [0.131, -63.598, 144.848, -60.585, -85.677, 7.615]
  MoveL 222 to (485.84, 896.21, 0) mm, rotated rx 0 ry 90 rz -60.43 deg; joints [-0.068, -63.592, 144.833, -60.784, -85.699, 7.637]
  MoveL 223 to (486.44, 899.62, 0) mm, rotated rx 0 ry 90 rz -60.43 deg; joints [-0.264, -63.573, 144.788, -60.98, -85.713, 7.675]
  MoveL 224 to (487.43, 902.93, 0) mm, rotated rx 0 ry 90 rz -60.43 deg; joints [-0.454, -63.542, 144.714, -61.172, -85.717, 7.727]
  MoveL 225 to (488.79, 906.09, 0) mm, rotated rx 0 ry 90 rz -60.43 deg; joints [-0.635, -63.499, 144.611, -61.355, -85.713, 7.793]
  MoveL 226 to (490.53, 909.06, 0) mm, rotated rx 0 ry 90 rz -60.43 deg; joints [-0.804, -63.445, 144.48, -61.528, -85.699, 7.873]
  MoveL 227 to (492.63, 911.8, 0) mm, rotated rx 0 ry 90 rz -60.43 deg; joints [-0.958, -63.379, 144.322, -61.688, -85.677, 7.966]
  MoveL 228 to (495.07, 914.25, 0) mm, rotated rx 0 ry 90 rz -60.43 deg; joints [-1.096, -63.302, 144.138, -61.832, -85.645, 8.071]
  MoveL 229 to (497.86, 916.38, 0) mm, rotated rx 0 ry 90 rz -60.43 deg; joints [-1.214, -63.215, 143.929, -61.957, -85.604, 8.188]
  MoveL 230 to (650.74, 1017.42, 0) mm, rotated rx 0 ry 90 rz -60.43 deg; joints [-6.018, -57.966, 131.867, -67.274, -83.638, 14.819]
  MoveL 231 to (650.74, 1065.95, 0) mm, rotated rx 0 ry 90 rz -60.43 deg; joints [-8.375, -57.753, 131.393, -69.589, -84.154, 15.307]
  MoveL 232 to (447.54, 931.66, 0) mm, rotated rx 0 ry 90 rz -60.43 deg; joints [-2.19, -64.721, 147.592, -62.8, -86.728, 6.338]
  MoveL 233 to (447.54, 765.88, 0) mm, rotated rx 0 ry 90 rz -60.43 deg; joints [7.678, -64.485, 147.009, -52.986, -85.483, 5.963]
  MoveL 234 to (788.26, 765.88, 0) mm, rotated rx 0 ry 90 rz -60.43 deg; joints [5.679, -52.932, 120.844, -56.78, -77.465, 18.335]
  MoveL 235 to (1064.06, 927.56, 0) mm, rotated rx 0 ry 90 rz -60.43 deg; joints [-1.184, -41.461, 96.59, -66.089, -74.227, 31.511]
  Set speed (60.0 mm/s)
  MoveL 236 to (1062.04, 930.4, 0) mm, rotated rx 0 ry 90 rz -60.43 deg; joints [-1.289, -41.555, 96.784, -66.155, -74.323, 31.44]
  MoveL 237 to (1059.84, 933.08, 0) mm, rotated rx 0 ry 90 rz -60.43 deg; joints [-1.389, -41.656, 96.996, -66.216, -74.419, 31.36]
  MoveL 238 to (1057.47, 935.61, 0) mm, rotated rx 0 ry 90 rz -60.43 deg; joints [-1.483, -41.766, 97.224, -66.269, -74.516, 31.269]
  MoveL 239 to (1054.94, 937.97, 0) mm, rotated rx 0 ry 90 rz -60.43 deg; joints [-1.572, -41.882, 97.467, -66.316, -74.613, 31.17]
  MoveL 240 to (1052.26, 940.17, 0) mm, rotated rx 0 ry 90 rz -60.43 deg; joints [-1.655, -42.006, 97.725, -66.356, -74.71, 31.062]
  MoveL 241 to (1049.45, 942.19, 0) mm, rotated rx 0 ry 90 rz -60.43 deg; joints [-1.732, -42.135, 97.995, -66.39, -74.806, 30.947]
  MoveL 242 to (1046.51, 944.04, 0) mm, rotated rx 0 ry 90 rz -60.43 deg; joints [-1.803, -42.27, 98.277, -66.416, -74.901, 30.824]
  MoveL 243 to (1043.45, 945.7, 0) mm, rotated rx 0 ry 90 rz -60.43 deg; joints [-1.868, -42.411, 98.57, -66.436, -74.996, 30.694]
  MoveL 244 to (1040.31, 947.17, 0) mm, rotated rx 0 ry 90 rz -60.43 deg; joints [-1.926, -42.555, 98.871, -66.45, -75.088, 30.559]
  MoveL 245 to (1037.1, 948.45, 0) mm, rotated rx 0 ry 90 rz -60.43 deg; joints [-1.977, -42.702, 99.179, -66.456, -75.178, 30.418]
  MoveL 246 to (1033.82, 949.53, 0) mm, rotated rx 0 ry 90 rz -60.43 deg; joints [-2.022, -42.853, 99.493, -66.456, -75.266, 30.273]
  MoveL 247 to (1030.48, 950.42, 0) mm, rotated rx 0 ry 90 rz -60.43 deg; joints [-2.059, -43.005, 99.812, -66.45, -75.351, 30.124]
  MoveL 248 to (1027.09, 951.11, 0) mm, rotated rx 0 ry 90 rz -60.43 deg; joints [-2.089, -43.16, 100.135, -66.436, -75.434, 29.971]
  MoveL 249 to (1023.67, 951.61, 0) mm, rotated rx 0 ry 90 rz -60.43 deg; joints [-2.112, -43.316, 100.462, -66.417, -75.513, 29.814]
  MoveL 250 to (1020.23, 951.9, 0) mm, rotated rx 0 ry 90 rz -60.43 deg; joints [-2.128, -43.474, 100.791, -66.39, -75.59, 29.656]
  MoveL 251 to (1016.77, 952, 0) mm, rotated rx 0 ry 90 rz -60.43 deg; joints [-2.137, -43.631, 101.121, -66.358, -75.663, 29.495]
  MoveL 252 to (920.39, 952, 0) mm, rotated rx 0 ry 90 rz -60.43 deg; joints [-2.281, -47.843, 109.98, -65.481, -77.626, 25.164]
  MoveL 253 to (920.39, 990.1, 0) mm, rotated rx 0 ry 90 rz -60.43 deg; joints [-3.802, -47.758, 109.801, -66.906, -78.24, 25.547]
  MoveL 254 to (1071.25, 990.1, 0) mm, rotated rx 0 ry 90 rz -60.43 deg; joints [-3.44, -40.996, 95.621, -68.199, -75.228, 32.515]
  MoveL 255 to (1171.98, 837.7, 0) mm, rotated rx 0 ry 90 rz -60.43 deg; joints [1.951, -35.964, 85.187, -65.087, -70.033, 36.324]
  MoveL 256 to (1123.45, 837.7, 0) mm, rotated rx 0 ry 90 rz -60.43 deg; joints [2.009, -38.506, 90.447, -64.171, -71.165, 33.703]
  MoveL 257 to (1064.06, 927.56, 0) mm, rotated rx 0 ry 90 rz -60.43 deg; joints [-1.184, -41.461, 96.59, -66.089, -74.227, 31.511]
  MoveL 258 to (970.82, 819.19, 0) mm, rotated rx 0 ry 90 rz -60.43 deg; joints [2.931, -45.645, 105.345, -61.185, -74.27, 26.235]
  Set speed (60.0 mm/s)
  MoveL 259 to (971.42, 822.6, 0) mm, rotated rx 0 ry 90 rz -60.43 deg; joints [2.798, -45.626, 105.306, -61.314, -74.319, 26.288]
  MoveL 260 to (972.4, 825.91, 0) mm, rotated rx 0 ry 90 rz -60.43 deg; joints [2.668, -45.59, 105.229, -61.444, -74.357, 26.357]
  MoveL 261 to (973.77, 829.08, 0) mm, rotated rx 0 ry 90 rz -60.43 deg; joints [2.544, -45.536, 105.117, -61.575, -74.384, 26.442]
  MoveL 262 to (975.51, 832.05, 0) mm, rotated rx 0 ry 90 rz -60.43 deg; joints [2.427, -45.466, 104.968, -61.703, -74.4, 26.542]
  MoveL 263 to (977.6, 834.78, 0) mm, rotated rx 0 ry 90 rz -60.43 deg; joints [2.318, -45.379, 104.785, -61.827, -74.403, 26.657]
  MoveL 264 to (980.05, 837.24, 0) mm, rotated rx 0 ry 90 rz -60.43 deg; joints [2.22, -45.275, 104.568, -61.946, -74.394, 26.786]
  MoveL 265 to (982.84, 839.37, 0) mm, rotated rx 0 ry 90 rz -60.43 deg; joints [2.134, -45.156, 104.317, -62.058, -74.371, 26.928]
  MoveL 266 to (1034.12, 873.26, 0) mm, rotated rx 0 ry 90 rz -60.43 deg; joints [0.807, -42.876, 99.542, -63.906, -73.865, 29.572]
  MoveL 267 to (1034.12, 921.79, 0) mm, rotated rx 0 ry 90 rz -60.43 deg; joints [-0.993, -42.873, 99.535, -65.53, -74.758, 30.014]
  MoveL 268 to (932.52, 854.64, 0) mm, rotated rx 0 ry 90 rz -60.43 deg; joints [1.603, -47.355, 108.949, -61.98, -75.744, 24.832]
  MoveL 269 to (932.52, 688.86, 0) mm, rotated rx 0 ry 90 rz -60.43 deg; joints [8.131, -46.754, 107.681, -55.958, -72.712, 23.744]
  MoveL 270 to (1155.67, 688.86, 0) mm, rotated rx 0 ry 90 rz -60.43 deg; joints [7.054, -36.211, 85.696, -60.528, -67.197, 34.442]
  MoveL 271 to (1193.77, 739.82, 0) mm, rotated rx 0 ry 90 rz -60.43 deg; joints [5.204, -34.429, 82.018, -62.857, -67.376, 36.882]
  MoveL 272 to (996.02, 739.82, 0) mm, rotated rx 0 ry 90 rz -60.43 deg; joints [5.882, -44.258, 102.434, -58.825, -72.19, 26.818]
  MoveL 273 to (993.39, 739.97, 0) mm, rotated rx 0 ry 90 rz -60.43 deg; joints [5.887, -44.376, 102.682, -58.785, -72.255, 26.701]
  MoveL 274 to (990.83, 740.4, 0) mm, rotated rx 0 ry 90 rz -60.43 deg; joints [5.881, -44.493, 102.925, -58.756, -72.324, 26.588]
  MoveL 275 to (988.35, 741.11, 0) mm, rotated rx 0 ry 90 rz -60.43 deg; joints [5.863, -44.606, 103.164, -58.738, -72.396, 26.481]
  MoveL 276 to (985.96, 742.08, 0) mm, rotated rx 0 ry 90 rz -60.43 deg; joints [5.836, -44.717, 103.395, -58.731, -72.471, 26.38]
  MoveL 277 to (983.7, 743.29, 0) mm, rotated rx 0 ry 90 rz -60.43 deg; joints [5.799, -44.823, 103.617, -58.735, -72.548, 26.287]
  MoveL 278 to (981.56, 744.74, 0) mm, rotated rx 0 ry 90 rz -60.43 deg; joints [5.752, -44.924, 103.83, -58.749, -72.626, 26.2]
  MoveL 279 to (979.56, 746.41, 0) mm, rotated rx 0 ry 90 rz -60.43 deg; joints [5.696, -45.019, 104.03, -58.774, -72.705, 26.122]
  MoveL 280 to (977.73, 748.28, 0) mm, rotated rx 0 ry 90 rz -60.43 deg; joints [5.632, -45.108, 104.217, -58.808, -72.784, 26.052]
  MoveL 281 to (976.08, 750.33, 0) mm, rotated rx 0 ry 90 rz -60.43 deg; joints [5.56, -45.189, 104.388, -58.852, -72.862, 25.992]
  MoveL 282 to (974.65, 752.52, 0) mm, rotated rx 0 ry 90 rz -60.43 deg; joints [5.481, -45.262, 104.54, -58.905, -72.938, 25.942]
  MoveL 283 to (973.43, 754.82, 0) mm, rotated rx 0 ry 90 rz -60.43 deg; joints [5.398, -45.325, 104.673, -58.966, -73.01, 25.903]
  MoveL 284 to (972.42, 757.23, 0) mm, rotated rx 0 ry 90 rz -60.43 deg; joints [5.309, -45.379, 104.786, -59.033, -73.08, 25.874]
  MoveL 285 to (971.64, 759.72, 0) mm, rotated rx 0 ry 90 rz -60.43 deg; joints [5.216, -45.424, 104.88, -59.107, -73.145, 25.855]
  MoveL 286 to (971.07, 762.27, 0) mm, rotated rx 0 ry 90 rz -60.43 deg; joints [5.121, -45.459, 104.953, -59.188, -73.207, 25.847]
  MoveL 287 to (970.73, 764.86, 0) mm, rotated rx 0 ry 90 rz -60.43 deg; joints [5.022, -45.484, 105.006, -59.273, -73.264, 25.849]
  MoveL 288 to (970.62, 767.48, 0) mm, rotated rx 0 ry 90 rz -60.43 deg; joints [4.922, -45.499, 105.037, -59.363, -73.316, 25.861]
  MoveL 289 to (970.62, 815.73, 0) mm, rotated rx 0 ry 90 rz -60.43 deg; joints [3.065, -45.646, 105.347, -61.06, -74.212, 26.2]
  MoveL 290 to (970.82, 819.19, 0) mm, rotated rx 0 ry 90 rz -60.43 deg; joints [2.931, -45.645, 105.345, -61.185, -74.27, 26.235]
  MoveL 291 to (868.9, 817.19, 0) mm, rotated rx 0 ry 90 rz -60.43 deg; joints [3.23, -49.922, 114.394, -59.819, -76.499, 21.872]
  Set speed (60.0 mm/s)
  MoveL 292 to (868.56, 819.78, 0) mm, rotated rx 0 ry 90 rz -60.43 deg; joints [3.123, -49.942, 114.436, -59.916, -76.55, 21.876]
  MoveL 293 to (867.99, 822.33, 0) mm, rotated rx 0 ry 90 rz -60.43 deg; joints [3.019, -49.97, 114.496, -60.009, -76.605, 21.871]
  MoveL 294 to (867.21, 824.82, 0) mm, rotated rx 0 ry 90 rz -60.43 deg; joints [2.917, -50.007, 114.575, -60.097, -76.663, 21.856]
  MoveL 295 to (866.2, 827.22, 0) mm, rotated rx 0 ry 90 rz -60.43 deg; joints [2.82, -50.053, 114.672, -60.18, -76.725, 21.832]
  MoveL 296 to (864.98, 829.53, 0) mm, rotated rx 0 ry 90 rz -60.43 deg; joints [2.726, -50.106, 114.786, -60.257, -76.79, 21.798]
  MoveL 297 to (863.55, 831.72, 0) mm, rotated rx 0 ry 90 rz -60.43 deg; joints [2.638, -50.168, 114.918, -60.327, -76.858, 21.755]
  MoveL 298 to (861.9, 833.77, 0) mm, rotated rx 0 ry 90 rz -60.43 deg; joints [2.556, -50.238, 115.067, -60.389, -76.927, 21.702]
  MoveL 299 to (860.07, 835.64, 0) mm, rotated rx 0 ry 90 rz -60.43 deg; joints [2.481, -50.315, 115.231, -60.443, -76.998, 21.64]
  MoveL 300 to (858.07, 837.31, 0) mm, rotated rx 0 ry 90 rz -60.43 deg; joints [2.415, -50.398, 115.408, -60.487, -77.069, 21.57]
  MoveL 301 to (855.93, 838.76, 0) mm, rotated rx 0 ry 90 rz -60.43 deg; joints [2.358, -50.486, 115.596, -60.521, -77.139, 21.493]
  MoveL 302 to (853.67, 839.97, 0) mm, rotated rx 0 ry 90 rz -60.43 deg; joints [2.311, -50.579, 115.794, -60.545, -77.208, 21.409]
  MoveL 303 to (851.28, 840.94, 0) mm, rotated rx 0 ry 90 rz -60.43 deg; joints [2.274, -50.676, 116.001, -60.559, -77.275, 21.319]
  MoveL 304 to (848.8, 841.65, 0) mm, rotated rx 0 ry 90 rz -60.43 deg; joints [2.249, -50.775, 116.214, -60.561, -77.34, 21.223]
  MoveL 305 to (846.24, 842.08, 0) mm, rotated rx 0 ry 90 rz -60.43 deg; joints [2.235, -50.878, 116.433, -60.552, -77.402, 21.122]
  MoveL 306 to (843.62, 842.23, 0) mm, rotated rx 0 ry 90 rz -60.43 deg; joints [2.233, -50.983, 116.657, -60.53, -77.462, 21.016]
  MoveL 307 to (685.05, 842.23, 0) mm, rotated rx 0 ry 90 rz -60.43 deg; joints [2.529, -56.941, 129.592, -59.088, -80.882, 14.823]
  MoveL 308 to (723.15, 893.18, 0) mm, rotated rx 0 ry 90 rz -60.43 deg; joints [0.085, -55.609, 126.66, -61.696, -80.754, 16.613]
  MoveL 309 to (907.12, 893.18, 0) mm, rotated rx 0 ry 90 rz -60.43 deg; joints [0.074, -48.445, 111.256, -63.149, -76.937, 24.059]
  MoveL 310 to (907.12, 727.4, 0) mm, rotated rx 0 ry 90 rz -60.43 deg; joints [6.744, -48.033, 110.383, -56.934, -74.048, 22.887]
  MoveL 311 to (703.92, 593.11, 0) mm, rotated rx 0 ry 90 rz -60.43 deg; joints [13.963, -54.957, 125.235, -48.192, -76.56, 14.568]
  MoveL 312 to (703.92, 641.64, 0) mm, rotated rx 0 ry 90 rz -60.43 deg; joints [11.787, -55.355, 126.105, -50.27, -77.417, 14.688]
  MoveL 313 to (856.79, 742.68, 0) mm, rotated rx 0 ry 90 rz -60.43 deg; joints [6.358, -50.158, 114.897, -56.76, -75.498, 20.912]
  MoveL 314 to (859.58, 744.81, 0) mm, rotated rx 0 ry 90 rz -60.43 deg; joints [6.257, -50.056, 114.678, -56.883, -75.471, 21.036]
  MoveL 315 to (862.03, 747.26, 0) mm, rotated rx 0 ry 90 rz -60.43 deg; joints [6.145, -49.968, 114.492, -57.013, -75.457, 21.149]
  MoveL 316 to (864.12, 750, 0) mm, rotated rx 0 ry 90 rz -60.43 deg; joints [6.023, -49.896, 114.337, -57.148, -75.457, 21.25]
  MoveL 317 to (865.86, 752.97, 0) mm, rotated rx 0 ry 90 rz -60.43 deg; joints [5.893, -49.838, 114.215, -57.287, -75.469, 21.338]
  MoveL 318 to (867.23, 756.13, 0) mm, rotated rx 0 ry 90 rz -60.43 deg; joints [5.757, -49.796, 114.125, -57.428, -75.493, 21.412]
  MoveL 319 to (868.21, 759.44, 0) mm, rotated rx 0 ry 90 rz -60.43 deg; joints [5.617, -49.77, 114.069, -57.57, -75.528, 21.472]
  MoveL 320 to (869.02, 766.32, 0) mm, rotated rx 0 ry 90 rz -60.43 deg; joints [5.33, -49.764, 114.057, -57.846, -75.629, 21.546]
  MoveL 321 to (869.02, 814.57, 0) mm, rotated rx 0 ry 90 rz -60.43 deg; joints [3.338, -49.912, 114.371, -59.718, -76.453, 21.859]
  MoveL 322 to (868.9, 817.19, 0) mm, rotated rx 0 ry 90 rz -60.43 deg; joints [3.23, -49.922, 114.394, -59.819, -76.499, 21.872]
  MoveL 323 to (226.56, 635.47, 0) mm, rotated rx -90 ry 80 rz -150.43 deg; joints [16.315, -67.747, 157.462, -44.114, -89.795, 10.199]
  Set speed (60.0 mm/s)
  MoveL 324 to (226.44, 638.09, 0) mm, rotated rx -90 ry 80 rz -150.43 deg; joints [16.141, -67.766, 157.521, -44.287, -89.825, 10.171]
  MoveL 325 to (226.44, 686.34, 0) mm, rotated rx -90 ry 70 rz -150.43 deg; joints [10.274, -65.239, 155.253, -50.155, -90.009, 19.99]
  MoveL 326 to (227.25, 693.22, 0) mm, rotated rx -90 ry 70 rz -150.43 deg; joints [9.808, -65.248, 155.282, -50.621, -90.022, 19.974]
  MoveL 327 to (228.23, 696.53, 0) mm, rotated rx -90 ry 70 rz -150.43 deg; joints [9.577, -65.239, 155.252, -50.851, -90.008, 19.99]
  MoveL 328 to (229.6, 699.69, 0) mm, rotated rx -90 ry 70 rz -150.43 deg; joints [9.352, -65.222, 155.193, -51.077, -89.982, 20.022]
  MoveL 329 to (231.33, 702.66, 0) mm, rotated rx -90 ry 70 rz -150.43 deg; joints [9.136, -65.197, 155.106, -51.292, -89.943, 20.071]
  MoveL 330 to (233.43, 705.4, 0) mm, rotated rx -90 ry 70 rz -150.43 deg; joints [8.933, -65.163, 154.989, -51.496, -89.892, 20.136]
  MoveL 331 to (235.88, 707.86, 0) mm, rotated rx -90 ry 70 rz -150.43 deg; joints [8.745, -65.12, 154.844, -51.684, -89.829, 20.217]
  MoveL 332 to (238.67, 709.99, 0) mm, rotated rx -90 ry 80 rz -150.43 deg; joints [11.041, -67.878, 157.877, -49.387, -89.999, 10.001]
  MoveL 333 to (391.54, 811.03, 0) mm, rotated rx 0 ry 90 rz -60.43 deg; joints [5.32, -66.231, 151.422, -55.203, -87.251, 3.947]
  MoveL 334 to (391.54, 859.56, 0) mm, rotated rx 0 ry 90 rz -60.43 deg; joints [2.252, -66.319, 151.653, -58.262, -87.541, 3.967]
  MoveL 335 to (188.34, 725.26, 0) mm, rotated rx -90 ry 60 rz -150.43 deg; joints [5.847, -62.315, 155.11, -54.613, -91.619, 27.722]
  MoveL 336 to (188.34, 559.48, 0) mm, rotated rx -90 ry 70 rz -150.43 deg; joints [19.222, -65.333, 155.577, -41.207, -90.184, 19.839]
  MoveL 337 to (450.69, 559.48, 0) mm, rotated rx 0 ry 90 rz -60.43 deg; joints [19.246, -62.92, 143.225, -41.592, -82.719, 6.418]
  MoveL 338 to (488.79, 610.43, 0) mm, rotated rx 0 ry 90 rz -60.43 deg; joints [15.898, -62.26, 141.667, -45.023, -82.47, 7.472]
  MoveL 339 to (251.84, 610.43, 0) mm, rotated rx -90 ry 80 rz -150.43 deg; joints [17.453, -67.013, 155.226, -42.99, -88.692, 11.219]
  MoveL 340 to (249.22, 610.58, 0) mm, rotated rx -90 ry 80 rz -150.43 deg; joints [17.496, -67.075, 155.408, -42.944, -88.779, 11.136]
  MoveL 341 to (246.66, 611.02, 0) mm, rotated rx -90 ry 80 rz -150.43 deg; joints [17.52, -67.137, 155.591, -42.919, -88.868, 11.053]
  MoveL 342 to (244.18, 611.72, 0) mm, rotated rx -90 ry 80 rz -150.43 deg; joints [17.525, -67.198, 155.774, -42.912, -88.957, 10.969]
  MoveL 343 to (241.79, 612.69, 0) mm, rotated rx -90 ry 80 rz -150.43 deg; joints [17.511, -67.259, 155.957, -42.925, -89.046, 10.887]
  MoveL 344 to (239.53, 613.91, 0) mm, rotated rx -90 ry 80 rz -150.43 deg; joints [17.479, -67.318, 156.136, -42.956, -89.135, 10.805]
  MoveL 345 to (237.39, 615.35, 0) mm, rotated rx -90 ry 80 rz -150.43 deg; joints [17.428, -67.376, 156.312, -43.005, -89.222, 10.726]
  MoveL 346 to (235.39, 617.02, 0) mm, rotated rx -90 ry 80 rz -150.43 deg; joints [17.36, -67.432, 156.483, -43.072, -89.306, 10.648]
  MoveL 347 to (233.56, 618.9, 0) mm, rotated rx -90 ry 80 rz -150.43 deg; joints [17.274, -67.486, 156.647, -43.157, -89.388, 10.574]
  MoveL 348 to (231.91, 620.95, 0) mm, rotated rx -90 ry 80 rz -150.43 deg; joints [17.173, -67.536, 156.801, -43.258, -89.465, 10.503]
  MoveL 349 to (230.48, 623.13, 0) mm, rotated rx -90 ry 80 rz -150.43 deg; joints [17.058, -67.582, 156.944, -43.372, -89.536, 10.438]
  MoveL 350 to (229.26, 625.44, 0) mm, rotated rx -90 ry 80 rz -150.43 deg; joints [16.93, -67.624, 157.075, -43.5, -89.602, 10.378]
  MoveL 351 to (228.25, 627.85, 0) mm, rotated rx -90 ry 80 rz -150.43 deg; joints [16.79, -67.662, 157.193, -43.639, -89.66, 10.324]
  MoveL 352 to (227.46, 630.33, 0) mm, rotated rx -90 ry 80 rz -150.43 deg; joints [16.64, -67.695, 157.297, -43.789, -89.712, 10.276]
  MoveL 353 to (226.9, 632.88, 0) mm, rotated rx -90 ry 80 rz -150.43 deg; joints [16.481, -67.724, 157.387, -43.948, -89.757, 10.234]
  MoveL 354 to (226.56, 635.47, 0) mm, rotated rx -90 ry 80 rz -150.43 deg; joints [16.315, -67.747, 157.462, -44.114, -89.795, 10.199]
  MoveL 355 to (571.07, 677.93, 0) mm, rotated rx 0 ry 90 rz -60.43 deg; joints [11.351, -60.171, 136.836, -49.851, -81.31, 10.154]
  Set speed (60.0 mm/s)
  MoveL 356 to (569.05, 680.77, 0) mm, rotated rx 0 ry 90 rz -60.43 deg; joints [11.226, -60.256, 137.029, -49.962, -81.402, 10.089]
  MoveL 357 to (566.85, 683.46, 0) mm, rotated rx 0 ry 90 rz -60.43 deg; joints [11.111, -60.345, 137.232, -50.064, -81.496, 10.018]
  MoveL 358 to (564.48, 685.98, 0) mm, rotated rx 0 ry 90 rz -60.43 deg; joints [11.006, -60.438, 137.446, -50.155, -81.591, 9.94]
  MoveL 359 to (561.95, 688.35, 0) mm, rotated rx 0 ry 90 rz -60.43 deg; joints [10.909, -60.535, 137.668, -50.237, -81.688, 9.856]
  MoveL 360 to (559.27, 690.54, 0) mm, rotated rx 0 ry 90 rz -60.43 deg; joints [10.822, -60.636, 137.899, -50.309, -81.786, 9.768]
  MoveL 361 to (556.46, 692.56, 0) mm, rotated rx 0 ry 90 rz -60.43 deg; joints [10.745, -60.74, 138.137, -50.371, -81.884, 9.674]
  MoveL 362 to (553.52, 694.41, 0) mm, rotated rx 0 ry 90 rz -60.43 deg; joints [10.678, -60.846, 138.382, -50.423, -81.984, 9.576]
  MoveL 363 to (550.46, 696.07, 0) mm, rotated rx 0 ry 90 rz -60.43 deg; joints [10.622, -60.955, 138.632, -50.464, -82.083, 9.474]
  MoveL 364 to (547.32, 697.54, 0) mm, rotated rx 0 ry 90 rz -60.43 deg; joints [10.576, -61.065, 138.885, -50.494, -82.182, 9.368]
  MoveL 365 to (544.11, 698.82, 0) mm, rotated rx 0 ry 90 rz -60.43 deg; joints [10.54, -61.176, 139.141, -50.515, -82.28, 9.26]
  MoveL 366 to (540.83, 699.9, 0) mm, rotated rx 0 ry 90 rz -60.43 deg; joints [10.515, -61.287, 139.399, -50.524, -82.377, 9.149]
  MoveL 367 to (537.49, 700.79, 0) mm, rotated rx 0 ry 90 rz -60.43 deg; joints [10.501, -61.399, 139.659, -50.523, -82.473, 9.037]
  MoveL 368 to (534.1, 701.48, 0) mm, rotated rx 0 ry 90 rz -60.43 deg; joints [10.498, -61.511, 139.918, -50.512, -82.567, 8.922]
  MoveL 369 to (530.68, 701.98, 0) mm, rotated rx 0 ry 90 rz -60.43 deg; joints [10.505, -61.623, 140.178, -50.489, -82.66, 8.806]
  MoveL 370 to (527.24, 702.28, 0) mm, rotated rx 0 ry 90 rz -60.43 deg; joints [10.523, -61.734, 140.436, -50.457, -82.751, 8.689]
  MoveL 371 to (523.78, 702.38, 0) mm, rotated rx 0 ry 90 rz -60.43 deg; joints [10.552, -61.844, 140.692, -50.414, -82.84, 8.572]
  MoveL 372 to (361.71, 702.38, 0) mm, rotated rx 0 ry 90 rz -60.43 deg; joints [12.457, -66.579, 152.337, -48.05, -87.161, 3.154]
  MoveL 373 to (361.71, 740.48, 0) mm, rotated rx 0 ry 90 rz -60.43 deg; joints [10.049, -66.78, 152.871, -50.445, -87.508, 3.013]
  MoveL 374 to (578.26, 740.48, 0) mm, rotated rx 0 ry 90 rz -60.43 deg; joints [8.08, -60.286, 137.099, -53.087, -81.989, 10.51]
  MoveL 375 to (678.99, 588.08, 0) mm, rotated rx 0 ry 90 rz -60.43 deg; joints [14.471, -55.798, 127.075, -47.512, -77.106, 13.692]
  MoveL 376 to (630.46, 588.08, 0) mm, rotated rx 0 ry 90 rz -60.43 deg; joints [15.059, -57.48, 130.785, -46.602, -78.357, 12.048]
  MoveL 377 to (571.07, 677.93, 0) mm, rotated rx 0 ry 90 rz -60.43 deg; joints [11.351, -60.171, 136.836, -49.851, -81.31, 10.154]
  MoveL 378 to (437.55, 432.48, 0) mm, rotated rx 0 ry 90 rz -60.43 deg; joints [26.01, -61.753, 140.481, -34.941, -80.721, 6.428]
  Set speed (60.0 mm/s)
  MoveL 379 to (437.55, 470.58, 0) mm, rotated rx 0 ry 90 rz -60.43 deg; joints [24.121, -62.269, 141.689, -36.778, -81.491, 6.312]
  MoveL 380 to (247.79, 470.58, 0) mm, rotated rx 0 ry 90 rz -60.43 deg; joints [29.241, -67.226, 154.075, -31.226, -87.305, 1.633]
  MoveL 381 to (234.07, 472.17, 0) mm, rotated rx 0 ry 90 rz -60.43 deg; joints [29.597, -67.555, 154.984, -30.857, -87.792, 1.319]
  MoveL 382 to (227.45, 474.14, 0) mm, rotated rx 0 ry 90 rz -60.43 deg; joints [29.702, -67.726, 155.463, -30.746, -88.055, 1.157]
  MoveL 383 to (221.1, 476.88, 0) mm, rotated rx 0 ry 90 rz -60.43 deg; joints [29.754, -67.899, 155.953, -30.689, -88.326, 0.993]
  MoveL 384 to (215.11, 480.39, 0) mm, rotated rx 0 ry 90 rz -60.43 deg; joints [29.749, -68.071, 156.447, -30.69, -88.603, 0.829]
  MoveL 385 to (209.62, 484.61, 0) mm, rotated rx 0 ry 90 rz -60.43 deg; joints [29.684, -68.239, 156.935, -30.751, -88.879, 0.667]
  MoveL 386 to (204.72, 489.5, 0) mm, rotated rx 0 ry 90 rz -60.43 deg; joints [29.557, -68.4, 157.408, -30.875, -89.149, 0.509]
  MoveL 387 to (200.5, 495.02, 0) mm, rotated rx 0 ry 90 rz -60.43 deg; joints [29.366, -68.551, 157.861, -31.065, -89.408, 0.356]
  MoveL 388 to (73.96, 686.48, 0) mm, rotated rx -90 ry 30 rz -150.43 deg; joints [4.419, -47.946, 153.425, -56.983, -98.581, 47.069]
  MoveL 389 to (25.43, 686.48, 0) mm, rotated rx -90 ry 30 rz -150.43 deg; joints [4.69, -47.213, 156.606, -57.278, -100.774, 43.778]
  MoveL 390 to (193.3, 432.48, 0) mm, rotated rx -90 ry 80 rz -150.43 deg; joints [29.881, -66.572, 153.947, -30.574, -87.739, 11.335]
  MoveL 391 to (437.55, 432.48, 0) mm, rotated rx 0 ry 90 rz -60.43 deg; joints [26.01, -61.753, 140.481, -34.941, -80.721, 6.428]
  MoveL 392 to (528.52, 612.28, 0) mm, rotated rx 0 ry 90 rz -60.43 deg; joints [15.225, -61.042, 138.832, -45.859, -81.43, 8.73]
  Set speed (60.0 mm/s)
  MoveL 393 to (526.5, 615.11, 0) mm, rotated rx 0 ry 90 rz -60.43 deg; joints [15.107, -61.13, 139.035, -45.964, -81.528, 8.664]
  MoveL 394 to (524.3, 617.79, 0) mm, rotated rx 0 ry 90 rz -60.43 deg; joints [14.999, -61.222, 139.247, -46.059, -81.628, 8.592]
  MoveL 395 to (521.94, 620.32, 0) mm, rotated rx 0 ry 90 rz -60.43 deg; joints [14.901, -61.317, 139.469, -46.144, -81.729, 8.514]
  MoveL 396 to (519.41, 622.68, 0) mm, rotated rx 0 ry 90 rz -60.43 deg; joints [14.814, -61.416, 139.698, -46.218, -81.833, 8.432]
  MoveL 397 to (516.74, 624.87, 0) mm, rotated rx 0 ry 90 rz -60.43 deg; joints [14.736, -61.518, 139.934, -46.282, -81.937, 8.345]
  MoveL 398 to (513.93, 626.89, 0) mm, rotated rx 0 ry 90 rz -60.43 deg; joints [14.669, -61.623, 140.177, -46.335, -82.042, 8.253]
  MoveL 399 to (511, 628.74, 0) mm, rotated rx 0 ry 90 rz -60.43 deg; joints [14.612, -61.729, 140.425, -46.377, -82.148, 8.158]
  MoveL 400 to (507.91, 630.42, 0) mm, rotated rx 0 ry 90 rz -60.43 deg; joints [14.566, -61.839, 140.68, -46.409, -82.255, 8.057]
  MoveL 401 to (504.81, 631.87, 0) mm, rotated rx 0 ry 90 rz -60.43 deg; joints [14.532, -61.947, 140.932, -46.429, -82.359, 7.957]
  MoveL 402 to (501.59, 633.15, 0) mm, rotated rx 0 ry 90 rz -60.43 deg; joints [14.508, -62.057, 141.189, -46.438, -82.464, 7.852]
  MoveL 403 to (498.3, 634.24, 0) mm, rotated rx 0 ry 90 rz -60.43 deg; joints [14.496, -62.167, 141.447, -46.437, -82.567, 7.746]
  MoveL 404 to (494.96, 635.13, 0) mm, rotated rx 0 ry 90 rz -60.43 deg; joints [14.494, -62.277, 141.706, -46.424, -82.67, 7.637]
  MoveL 405 to (491.57, 635.82, 0) mm, rotated rx 0 ry 90 rz -60.43 deg; joints [14.504, -62.386, 141.964, -46.401, -82.771, 7.528]
  MoveL 406 to (488.14, 636.32, 0) mm, rotated rx 0 ry 90 rz -60.43 deg; joints [14.525, -62.495, 142.22, -46.366, -82.87, 7.418]
  MoveL 407 to (484.69, 636.62, 0) mm, rotated rx 0 ry 90 rz -60.43 deg; joints [14.557, -62.603, 142.474, -46.321, -82.967, 7.307]
  MoveL 408 to (481.23, 636.72, 0) mm, rotated rx 0 ry 90 rz -60.43 deg; joints [14.6, -62.709, 142.725, -46.265, -83.061, 7.196]
  MoveL 409 to (269.9, 636.72, 0) mm, rotated rx 0 ry 90 rz -60.43 deg; joints [18.316, -68.403, 157.419, -42.116, -89.27, 0.66]
  MoveL 410 to (269.9, 674.82, 0) mm, rotated rx -90 ry 80 rz -150.43 deg; joints [12.959, -67, 155.188, -47.484, -88.775, 11.336]
  MoveL 411 to (535.71, 674.82, 0) mm, rotated rx 0 ry 90 rz -60.43 deg; joints [11.887, -61.292, 139.41, -49.156, -82.165, 8.961]
  MoveL 412 to (636.44, 522.42, 0) mm, rotated rx 0 ry 90 rz -60.43 deg; joints [17.999, -56.611, 128.863, -43.823, -76.997, 12.186]
  MoveL 413 to (587.91, 522.42, 0) mm, rotated rx 0 ry 90 rz -60.43 deg; joints [18.74, -58.237, 132.473, -42.782, -78.294, 10.634]
  MoveL 414 to (528.52, 612.28, 0) mm, rotated rx 0 ry 90 rz -60.43 deg; joints [15.225, -61.042, 138.832, -45.859, -81.43, 8.73]
  MoveL 415 to (1077.92, 419.21, 0) mm, rotated rx 0 ry 90 rz -60.43 deg; joints [16.677, -37.309, 87.968, -51.067, -62.747, 29.546]
  Set speed (60.0 mm/s)
  MoveL 416 to (1116.02, 419.21, 0) mm, rotated rx 0 ry 90 rz -60.43 deg; joints [16.307, -35.352, 83.923, -52.291, -61.64, 31.566]
  MoveL 417 to (1116.02, 663.46, 0) mm, rotated rx 0 ry 90 rz -60.43 deg; joints [8.103, -38.099, 89.603, -58.853, -67.64, 32.19]
  MoveL 418 to (862.02, 663.46, 0) mm, rotated rx 0 ry 90 rz -60.43 deg; joints [9.577, -49.503, 113.502, -53.808, -73.932, 20.72]
  MoveL 419 to (862.02, 612.51, 0) mm, rotated rx 0 ry 90 rz -60.43 deg; joints [11.632, -49.12, 112.686, -51.903, -72.948, 20.507]
  MoveL 420 to (1027.12, 612.51, 0) mm, rotated rx 0 ry 90 rz -60.43 deg; joints [10.412, -42.008, 97.73, -55.28, -68.783, 27.576]
  MoveL 421 to (1032.37, 612.21, 0) mm, rotated rx 0 ry 90 rz -60.43 deg; joints [10.388, -41.762, 97.216, -55.389, -68.642, 27.821]
  MoveL 422 to (1037.49, 611.35, 0) mm, rotated rx 0 ry 90 rz -60.43 deg; joints [10.385, -41.515, 96.701, -55.478, -68.491, 28.058]
  MoveL 423 to (1042.45, 609.93, 0) mm, rotated rx 0 ry 90 rz -60.43 deg; joints [10.403, -41.27, 96.191, -55.547, -68.333, 28.287]
  MoveL 424 to (1047.22, 608, 0) mm, rotated rx 0 ry 90 rz -60.43 deg; joints [10.441, -41.028, 95.688, -55.597, -68.167, 28.507]
  MoveL 425 to (1051.75, 605.57, 0) mm, rotated rx 0 ry 90 rz -60.43 deg; joints [10.497, -40.792, 95.195, -55.629, -67.995, 28.714]
  MoveL 426 to (1056.03, 602.67, 0) mm, rotated rx 0 ry 90 rz -60.43 deg; joints [10.572, -40.562, 94.718, -55.642, -67.819, 28.909]
  MoveL 427 to (1060.02, 599.34, 0) mm, rotated rx 0 ry 90 rz -60.43 deg; joints [10.663, -40.341, 94.258, -55.636, -67.64, 29.089]
  MoveL 428 to (1063.69, 595.59, 0) mm, rotated rx 0 ry 90 rz -60.43 deg; joints [10.771, -40.131, 93.821, -55.612, -67.46, 29.253]
  MoveL 429 to (1066.98, 591.48, 0) mm, rotated rx 0 ry 90 rz -60.43 deg; joints [10.892, -39.934, 93.412, -55.57, -67.28, 29.398]
  MoveL 430 to (1069.85, 587.11, 0) mm, rotated rx 0 ry 90 rz -60.43 deg; joints [11.026, -39.754, 93.038, -55.511, -67.105, 29.523]
  MoveL 431 to (1072.29, 582.5, 0) mm, rotated rx 0 ry 90 rz -60.43 deg; joints [11.17, -39.591, 92.699, -55.436, -66.934, 29.627]
  MoveL 432 to (1074.3, 577.69, 0) mm, rotated rx 0 ry 90 rz -60.43 deg; joints [11.324, -39.446, 92.399, -55.346, -66.77, 29.709]
  MoveL 433 to (1075.88, 572.71, 0) mm, rotated rx 0 ry 90 rz -60.43 deg; joints [11.485, -39.321, 92.137, -55.241, -66.612, 29.77]
  MoveL 434 to (1077.01, 567.62, 0) mm, rotated rx 0 ry 90 rz -60.43 deg; joints [11.654, -39.214, 91.916, -55.122, -66.463, 29.809]
  MoveL 435 to (1077.69, 562.43, 0) mm, rotated rx 0 ry 90 rz -60.43 deg; joints [11.829, -39.128, 91.737, -54.99, -66.323, 29.826]
  MoveL 436 to (1077.92, 557.19, 0) mm, rotated rx 0 ry 90 rz -60.43 deg; joints [12.008, -39.062, 91.601, -54.846, -66.193, 29.821]
  MoveL 437 to (1077.92, 419.21, 0) mm, rotated rx 0 ry 90 rz -60.43 deg; joints [16.677, -37.309, 87.968, -51.067, -62.747, 29.546]
  MoveL 438 to (169.13, 240.44, 0) mm, rotated rx 0 ry 90 rz -60.43 deg; joints [43.929, -65.163, 148.693, -16.599, -83.797, 1.845]
  Set speed (60.0 mm/s)
  MoveL 439 to (165.77, 242.52, 0) mm, rotated rx 0 ry 90 rz -60.43 deg; joints [43.98, -65.274, 148.973, -16.543, -83.958, 1.791]
  MoveL 440 to (162.31, 244.16, 0) mm, rotated rx 0 ry 90 rz -60.43 deg; joints [44.055, -65.379, 149.237, -16.463, -84.108, 1.738]
  MoveL 441 to (158.78, 245.34, 0) mm, rotated rx 0 ry 90 rz -60.43 deg; joints [44.154, -65.475, 149.481, -16.359, -84.247, 1.686]
  MoveL 442 to (155.16, 246.02, 0) mm, rotated rx 0 ry 90 rz -60.43 deg; joints [44.279, -65.563, 149.704, -16.23, -84.373, 1.635]
  MoveL 443 to (151.46, 246.17, 0) mm, rotated rx 0 ry 90 rz -60.43 deg; joints [44.432, -65.641, 149.903, -16.073, -84.484, 1.586]
  MoveL 444 to (147.69, 245.75, 0) mm, rotated rx 0 ry 90 rz -60.43 deg; joints [44.614, -65.709, 150.076, -15.887, -84.581, 1.54]
  MoveL 445 to (143.86, 244.72, 0) mm, rotated rx 0 ry 90 rz -60.43 deg; joints [44.827, -65.766, 150.221, -15.671, -84.66, 1.496]
  MoveL 446 to (139.97, 243.06, 0) mm, rotated rx 0 ry 90 rz -60.43 deg; joints [45.071, -65.81, 150.335, -15.425, -84.721, 1.454]
  MoveL 447 to (136.02, 240.72, 0) mm, rotated rx 0 ry 90 rz -60.43 deg; joints [45.348, -65.842, 150.416, -15.145, -84.762, 1.416]
  MoveL 448 to (132.02, 237.68, 0) mm, rotated rx 0 ry 90 rz -60.43 deg; joints [45.658, -65.86, 150.462, -14.833, -84.781, 1.38]
  MoveL 449 to (127.98, 233.89, 0) mm, rotated rx 0 ry 90 rz -60.43 deg; joints [46.004, -65.863, 150.469, -14.486, -84.777, 1.347]
  MoveL 450 to (122.21, 227.21, 0) mm, rotated rx 0 ry 90 rz -60.43 deg; joints [46.551, -65.839, 150.408, -13.938, -84.728, 1.306]
  MoveL 451 to (117.01, 219.8, 0) mm, rotated rx 0 ry 90 rz -60.43 deg; joints [47.103, -65.787, 150.275, -13.385, -84.637, 1.274]
  MoveL 452 to (112.37, 212, 0) mm, rotated rx 0 ry 90 rz -60.43 deg; joints [47.642, -65.713, 150.087, -12.846, -84.513, 1.249]
  MoveL 453 to (108.32, 204.19, 0) mm, rotated rx 0 ry 90 rz -60.43 deg; joints [48.153, -65.626, 149.864, -12.336, -84.37, 1.229]
  MoveL 454 to (104.31, 195.46, 0) mm, rotated rx 0 ry 90 rz -60.43 deg; joints [48.695, -65.516, 149.583, -11.795, -84.192, 1.211]
  MoveL 455 to (100.58, 186.36, 0) mm, rotated rx 0 ry 90 rz -60.43 deg; joints [49.234, -65.389, 149.263, -11.257, -83.991, 1.194]
  MoveL 456 to (93.92, 167.42, 0) mm, rotated rx 0 ry 90 rz -60.43 deg; joints [50.289, -65.096, 148.524, -10.205, -83.532, 1.162]
  MoveL 457 to (88.29, 148.15, 0) mm, rotated rx 0 ry 90 rz -60.43 deg; joints [51.285, -64.763, 147.696, -9.212, -83.023, 1.129]
  MoveL 458 to (83.64, 129.34, 0) mm, rotated rx 0 ry 90 rz -60.43 deg; joints [52.196, -64.411, 146.827, -8.305, -82.494, 1.092]
  MoveL 459 to (82.2, 122.92, 0) mm, rotated rx 0 ry 90 rz -60.43 deg; joints [52.494, -64.285, 146.518, -8.007, -82.308, 1.079]
  MoveL 460 to (77.52, 99.15, 0) mm, rotated rx 0 ry 90 rz -60.43 deg; joints [53.547, -63.798, 145.331, -6.956, -81.594, 1.022]
  MoveL 461 to (73.6, 74.87, 0) mm, rotated rx 0 ry 90 rz -60.43 deg; joints [54.548, -63.266, 144.05, -5.957, -80.834, 0.952]
  MoveL 462 to (70.4, 50.34, 0) mm, rotated rx 0 ry 90 rz -60.43 deg; joints [55.488, -62.697, 142.697, -5.016, -80.037, 0.87]
  MoveL 463 to (67.87, 25.85, 0) mm, rotated rx 0 ry 90 rz -60.43 deg; joints [56.364, -62.1, 141.29, -4.137, -79.218, 0.775]
  MoveL 464 to (63.5, 25.44, 0) mm, rotated rx 0 ry 90 rz -60.43 deg; joints [56.577, -62.166, 141.445, -3.92, -79.304, 0.729]
  MoveL 465 to (25.4, 25.44, 0) mm, rotated rx 0 ry 90 rz -60.43 deg; joints [58.361, -62.813, 142.971, -2.098, -80.165, 0.359]
  MoveL 466 to (25.4, 591.47, 0) mm, rotated rx -90 ry 30 rz -150.43 deg; joints [11.444, -47.46, 155.737, -50.448, -101.877, 46.006]
  MoveL 467 to (434.22, 25.44, 0) mm, rotated rx 0 ry 90 rz -60.43 deg; joints [42.632, -53.736, 122.582, -18.993, -69.903, 6.745]
  MoveL 468 to (404.04, 32.53, 0) mm, rotated rx 0 ry 90 rz -60.43 deg; joints [43.326, -54.745, 124.772, -18.127, -70.946, 6.1]
  MoveL 469 to (373.28, 38.93, 0) mm, rotated rx 0 ry 90 rz -60.43 deg; joints [44.092, -55.725, 126.914, -17.205, -71.976, 5.473]
  MoveL 470 to (342.35, 44.38, 0) mm, rotated rx 0 ry 90 rz -60.43 deg; joints [44.929, -56.66, 128.971, -16.229, -72.974, 4.871]
  MoveL 471 to (311.63, 48.63, 0) mm, rotated rx 0 ry 90 rz -60.43 deg; joints [45.837, -57.534, 130.906, -15.199, -73.923, 4.303]
  MoveL 472 to (184.4, 224.78, 0) mm, rotated rx 0 ry 90 rz -60.43 deg; joints [43.97, -64.521, 147.098, -16.59, -82.882, 2.114]
  MoveL 473 to (178.62, 231.96, 0) mm, rotated rx 0 ry 90 rz -60.43 deg; joints [43.901, -64.792, 147.766, -16.646, -83.266, 2.008]
  MoveL 474 to (172.4, 237.96, 0) mm, rotated rx 0 ry 90 rz -60.43 deg; joints [43.9, -65.045, 148.396, -16.634, -83.628, 1.899]
  MoveL 475 to (169.13, 240.44, 0) mm, rotated rx 0 ry 90 rz -60.43 deg; joints [43.929, -65.163, 148.693, -16.599, -83.797, 1.845]
  MoveL 476 to (740.63, 520.58, 0) mm, rotated rx 0 ry 90 rz -60.43 deg; joints [16.663, -52.902, 120.778, -45.956, -74.218, 15.706]
  Set speed (60.0 mm/s)
  MoveL 477 to (743.25, 520.7, 0) mm, rotated rx 0 ry 90 rz -60.43 deg; joints [16.625, -52.807, 120.573, -46.016, -74.152, 15.799]
  MoveL 478 to (791.49, 520.7, 0) mm, rotated rx 0 ry 90 rz -60.43 deg; joints [16.041, -50.999, 116.691, -47.045, -72.893, 17.534]
  MoveL 479 to (798.37, 519.9, 0) mm, rotated rx 0 ry 90 rz -60.43 deg; joints [15.994, -50.727, 116.11, -47.162, -72.696, 17.785]
  MoveL 480 to (801.68, 518.91, 0) mm, rotated rx 0 ry 90 rz -60.43 deg; joints [15.995, -50.589, 115.815, -47.197, -72.589, 17.905]
  MoveL 481 to (804.85, 517.54, 0) mm, rotated rx 0 ry 90 rz -60.43 deg; joints [16.014, -50.452, 115.523, -47.214, -72.478, 18.019]
  MoveL 482 to (807.82, 515.81, 0) mm, rotated rx 0 ry 90 rz -60.43 deg; joints [16.049, -50.318, 115.238, -47.214, -72.364, 18.125]
  MoveL 483 to (810.55, 513.71, 0) mm, rotated rx 0 ry 90 rz -60.43 deg; joints [16.102, -50.189, 114.963, -47.196, -72.249, 18.222]
  MoveL 484 to (813.01, 511.27, 0) mm, rotated rx 0 ry 90 rz -60.43 deg; joints [16.171, -50.067, 114.701, -47.159, -72.133, 18.307]
  MoveL 485 to (815.14, 508.48, 0) mm, rotated rx 0 ry 90 rz -60.43 deg; joints [16.257, -49.953, 114.458, -47.104, -72.018, 18.38]
  MoveL 486 to (916.18, 355.6, 0) mm, rotated rx 0 ry 90 rz -60.43 deg; joints [20.713, -43.771, 101.414, -44.519, -65.689, 22.04]
  MoveL 487 to (964.71, 355.6, 0) mm, rotated rx 0 ry 90 rz -60.43 deg; joints [20.087, -41.659, 97.001, -45.917, -64.314, 24.11]
  MoveL 488 to (830.41, 558.8, 0) mm, rotated rx 0 ry 90 rz -60.43 deg; joints [14.077, -49.889, 114.322, -49.287, -72.67, 19.094]
  MoveL 489 to (664.63, 558.8, 0) mm, rotated rx 0 ry 90 rz -60.43 deg; joints [15.968, -56.022, 127.566, -45.973, -76.941, 13.157]
  MoveL 490 to (664.63, 254, 0) mm, rotated rx 0 ry 90 rz -60.43 deg; joints [28.614, -51.635, 118.054, -34.094, -70.127, 12.958]
  MoveL 491 to (715.59, 254, 0) mm, rotated rx 0 ry 90 rz -60.43 deg; joints [27.604, -49.843, 114.225, -35.58, -68.695, 14.57]
  MoveL 492 to (715.59, 495.3, 0) mm, rotated rx 0 ry 90 rz -60.43 deg; joints [18.058, -53.526, 122.126, -44.413, -74.362, 14.794]
  MoveL 493 to (715.73, 497.93, 0) mm, rotated rx 0 ry 90 rz -60.43 deg; joints [17.945, -53.551, 122.181, -44.521, -74.412, 14.803]
  MoveL 494 to (716.17, 500.49, 0) mm, rotated rx 0 ry 90 rz -60.43 deg; joints [17.831, -53.565, 122.212, -44.632, -74.453, 14.822]
  MoveL 495 to (716.88, 502.97, 0) mm, rotated rx 0 ry 90 rz -60.43 deg; joints [17.716, -53.568, 122.219, -44.746, -74.484, 14.85]
  MoveL 496 to (717.84, 505.35, 0) mm, rotated rx 0 ry 90 rz -60.43 deg; joints [17.602, -53.561, 122.202, -44.862, -74.507, 14.887]
  MoveL 497 to (719.06, 507.62, 0) mm, rotated rx 0 ry 90 rz -60.43 deg; joints [17.49, -53.543, 122.163, -44.979, -74.522, 14.932]
  MoveL 498 to (720.51, 509.76, 0) mm, rotated rx 0 ry 90 rz -60.43 deg; joints [17.38, -53.515, 122.103, -45.096, -74.527, 14.986]
  MoveL 499 to (722.17, 511.75, 0) mm, rotated rx 0 ry 90 rz -60.43 deg; joints [17.273, -53.477, 122.021, -45.211, -74.523, 15.047]
  MoveL 500 to (724.05, 513.58, 0) mm, rotated rx 0 ry 90 rz -60.43 deg; joints [17.171, -53.429, 121.918, -45.325, -74.511, 15.115]
  MoveL 501 to (726.1, 515.23, 0) mm, rotated rx 0 ry 90 rz -60.43 deg; joints [17.075, -53.373, 121.797, -45.434, -74.491, 15.189]
  MoveL 502 to (728.29, 516.66, 0) mm, rotated rx 0 ry 90 rz -60.43 deg; joints [16.985, -53.31, 121.659, -45.538, -74.462, 15.267]
  MoveL 503 to (730.59, 517.89, 0) mm, rotated rx 0 ry 90 rz -60.43 deg; joints [16.904, -53.239, 121.507, -45.636, -74.426, 15.35]
  MoveL 504 to (733, 518.89, 0) mm, rotated rx 0 ry 90 rz -60.43 deg; joints [16.831, -53.163, 121.341, -45.727, -74.384, 15.435]
  MoveL 505 to (735.49, 519.68, 0) mm, rotated rx 0 ry 90 rz -60.43 deg; joints [16.766, -53.08, 121.164, -45.811, -74.335, 15.524]
  MoveL 506 to (738.03, 520.24, 0) mm, rotated rx 0 ry 90 rz -60.43 deg; joints [16.71, -52.993, 120.976, -45.887, -74.279, 15.614]
  MoveL 507 to (740.63, 520.58, 0) mm, rotated rx 0 ry 90 rz -60.43 deg; joints [16.663, -52.902, 120.778, -45.956, -74.218, 15.706]
  MoveL 508 to (531.29, 471.54, 0) mm, rotated rx 0 ry 90 rz -60.43 deg; joints [22.124, -59.45, 135.198, -39.179, -78.861, 8.947]
  Set speed (60.0 mm/s)
  MoveL 509 to (529.27, 474.38, 0) mm, rotated rx 0 ry 90 rz -60.43 deg; joints [22.028, -59.549, 135.423, -39.259, -78.973, 8.885]
  MoveL 510 to (527.07, 477.06, 0) mm, rotated rx 0 ry 90 rz -60.43 deg; joints [21.943, -59.652, 135.656, -39.329, -79.087, 8.817]
  MoveL 511 to (524.7, 479.59, 0) mm, rotated rx 0 ry 90 rz -60.43 deg; joints [21.868, -59.758, 135.896, -39.388, -79.202, 8.745]
  MoveL 512 to (522.17, 481.95, 0) mm, rotated rx 0 ry 90 rz -60.43 deg; joints [21.804, -59.867, 136.143, -39.436, -79.319, 8.668]
  MoveL 513 to (519.49, 484.15, 0) mm, rotated rx 0 ry 90 rz -60.43 deg; joints [21.75, -59.977, 136.395, -39.474, -79.436, 8.586]
  MoveL 514 to (516.68, 486.17, 0) mm, rotated rx 0 ry 90 rz -60.43 deg; joints [21.707, -60.09, 136.651, -39.5, -79.553, 8.501]
  MoveL 515 to (513.74, 488.02, 0) mm, rotated rx 0 ry 90 rz -60.43 deg; joints [21.674, -60.204, 136.911, -39.516, -79.671, 8.413]
  MoveL 516 to (510.68, 489.68, 0) mm, rotated rx 0 ry 90 rz -60.43 deg; joints [21.652, -60.319, 137.174, -39.521, -79.788, 8.321]
  MoveL 517 to (507.54, 491.15, 0) mm, rotated rx 0 ry 90 rz -60.43 deg; joints [21.641, -60.434, 137.437, -39.515, -79.903, 8.228]
  MoveL 518 to (504.33, 492.42, 0) mm, rotated rx 0 ry 90 rz -60.43 deg; joints [21.641, -60.549, 137.699, -39.499, -80.017, 8.132]
  MoveL 519 to (501.05, 493.51, 0) mm, rotated rx 0 ry 90 rz -60.43 deg; joints [21.652, -60.663, 137.961, -39.471, -80.13, 8.035]
  MoveL 520 to (497.71, 494.4, 0) mm, rotated rx 0 ry 90 rz -60.43 deg; joints [21.673, -60.776, 138.22, -39.434, -80.24, 7.937]
  MoveL 521 to (494.32, 495.09, 0) mm, rotated rx 0 ry 90 rz -60.43 deg; joints [21.706, -60.888, 138.478, -39.386, -80.348, 7.838]
  MoveL 522 to (490.9, 495.58, 0) mm, rotated rx 0 ry 90 rz -60.43 deg; joints [21.748, -60.998, 138.732, -39.327, -80.453, 7.738]
  MoveL 523 to (487.46, 495.88, 0) mm, rotated rx 0 ry 90 rz -60.43 deg; joints [21.802, -61.106, 138.981, -39.259, -80.555, 7.639]
  MoveL 524 to (484, 495.98, 0) mm, rotated rx 0 ry 90 rz -60.43 deg; joints [21.865, -61.213, 139.226, -39.18, -80.655, 7.539]
  MoveL 525 to (289.09, 495.98, 0) mm, rotated rx 0 ry 90 rz -60.43 deg; joints [26.525, -66.568, 152.307, -33.977, -86.465, 2.38]
  MoveL 526 to (289.09, 534.08, 0) mm, rotated rx 0 ry 90 rz -60.43 deg; joints [24.298, -67.007, 153.481, -36.182, -87.153, 2.081]
  MoveL 527 to (538.48, 534.08, 0) mm, rotated rx 0 ry 90 rz -60.43 deg; joints [18.99, -59.963, 136.362, -42.249, -79.846, 9.097]
  MoveL 528 to (639.21, 381.68, 0) mm, rotated rx 0 ry 90 rz -60.43 deg; joints [24.063, -54.67, 124.611, -38.093, -73.967, 12.217]
  MoveL 529 to (590.68, 381.68, 0) mm, rotated rx 0 ry 90 rz -60.43 deg; joints [24.996, -56.287, 128.149, -36.823, -75.306, 10.753]
  MoveL 530 to (531.29, 471.54, 0) mm, rotated rx 0 ry 90 rz -60.43 deg; joints [22.124, -59.45, 135.198, -39.179, -78.861, 8.947]
  MoveL 531 to (715.95, 227.1, 0) mm, rotated rx 0 ry 90 rz -60.43 deg; joints [28.575, -49.314, 113.1, -34.705, -67.963, 14.566]
  Set speed (60.0 mm/s)
  MoveL 532 to (713.33, 226.99, 0) mm, rotated rx 0 ry 90 rz -60.43 deg; joints [28.631, -49.406, 113.295, -34.623, -68.034, 14.481]
  MoveL 533 to (665.08, 226.99, 0) mm, rotated rx 0 ry 90 rz -60.43 deg; joints [29.61, -51.101, 116.911, -33.184, -69.396, 12.96]
  MoveL 534 to (658.2, 227.79, 0) mm, rotated rx 0 ry 90 rz -60.43 deg; joints [29.725, -51.353, 117.45, -33.005, -69.611, 12.751]
  MoveL 535 to (654.89, 228.77, 0) mm, rotated rx 0 ry 90 rz -60.43 deg; joints [29.759, -51.486, 117.734, -32.94, -69.731, 12.651]
  MoveL 536 to (651.73, 230.14, 0) mm, rotated rx 0 ry 90 rz -60.43 deg; joints [29.775, -51.62, 118.023, -32.892, -69.856, 12.556]
  MoveL 537 to (648.76, 231.88, 0) mm, rotated rx 0 ry 90 rz -60.43 deg; joints [29.774, -51.755, 118.312, -32.863, -69.986, 12.467]
  MoveL 538 to (646.02, 233.97, 0) mm, rotated rx 0 ry 90 rz -60.43 deg; joints [29.754, -51.889, 118.599, -32.853, -70.119, 12.386]
  MoveL 539 to (643.57, 236.42, 0) mm, rotated rx 0 ry 90 rz -60.43 deg; joints [29.715, -52.019, 118.879, -32.865, -70.253, 12.313]
  MoveL 540 to (641.44, 239.21, 0) mm, rotated rx 0 ry 90 rz -60.43 deg; joints [29.656, -52.145, 119.149, -32.898, -70.387, 12.25]
  MoveL 541 to (540.39, 392.09, 0) mm, rotated rx 0 ry 90 rz -60.43 deg; joints [25.577, -58.058, 132.071, -35.918, -76.937, 9.298]
  MoveL 542 to (491.86, 392.09, 0) mm, rotated rx 0 ry 90 rz -60.43 deg; joints [26.648, -59.555, 135.436, -34.598, -78.302, 7.962]
  MoveL 543 to (626.16, 188.89, 0) mm, rotated rx 0 ry 90 rz -60.43 deg; joints [31.853, -51.653, 118.092, -30.719, -69.45, 11.782]
  MoveL 544 to (791.94, 188.89, 0) mm, rotated rx 0 ry 90 rz -60.43 deg; joints [28.467, -45.719, 105.501, -35.831, -64.723, 17.135]
  MoveL 545 to (791.94, 493.69, 0) mm, rotated rx 0 ry 90 rz -60.43 deg; joints [17.128, -50.675, 115.999, -46.043, -72.312, 17.49]
  MoveL 546 to (740.99, 493.69, 0) mm, rotated rx 0 ry 90 rz -60.43 deg; joints [17.782, -52.582, 120.089, -44.911, -73.657, 15.67]
  MoveL 547 to (740.99, 252.39, 0) mm, rotated rx 0 ry 90 rz -60.43 deg; joints [27.183, -48.891, 112.201, -36.268, -67.936, 15.409]
  MoveL 548 to (740.84, 249.76, 0) mm, rotated rx 0 ry 90 rz -60.43 deg; joints [27.28, -48.847, 112.107, -36.178, -67.87, 15.402]
  MoveL 549 to (740.41, 247.2, 0) mm, rotated rx 0 ry 90 rz -60.43 deg; joints [27.381, -48.814, 112.038, -36.082, -67.813, 15.386]
  MoveL 550 to (739.7, 244.72, 0) mm, rotated rx 0 ry 90 rz -60.43 deg; joints [27.484, -48.793, 111.993, -35.98, -67.767, 15.361]
  MoveL 551 to (738.73, 242.34, 0) mm, rotated rx 0 ry 90 rz -60.43 deg; joints [27.588, -48.783, 111.971, -35.875, -67.73, 15.327]
  MoveL 552 to (737.52, 240.07, 0) mm, rotated rx 0 ry 90 rz -60.43 deg; joints [27.693, -48.784, 111.973, -35.765, -67.703, 15.285]
  MoveL 553 to (736.07, 237.93, 0) mm, rotated rx 0 ry 90 rz -60.43 deg; joints [27.797, -48.796, 111.998, -35.653, -67.687, 15.235]
  MoveL 554 to (734.4, 235.93, 0) mm, rotated rx 0 ry 90 rz -60.43 deg; joints [27.9, -48.818, 112.046, -35.539, -67.68, 15.178]
  MoveL 555 to (732.53, 234.1, 0) mm, rotated rx 0 ry 90 rz -60.43 deg; joints [28.002, -48.851, 112.116, -35.425, -67.683, 15.115]
  MoveL 556 to (730.48, 232.45, 0) mm, rotated rx 0 ry 90 rz -60.43 deg; joints [28.1, -48.894, 112.206, -35.311, -67.697, 15.046]
  MoveL 557 to (728.29, 231.02, 0) mm, rotated rx 0 ry 90 rz -60.43 deg; joints [28.194, -48.945, 112.316, -35.199, -67.72, 14.973]
  MoveL 558 to (725.98, 229.8, 0) mm, rotated rx 0 ry 90 rz -60.43 deg; joints [28.282, -49.005, 112.443, -35.091, -67.752, 14.896]
  MoveL 559 to (723.58, 228.79, 0) mm, rotated rx 0 ry 90 rz -60.43 deg; joints [28.365, -49.072, 112.586, -34.987, -67.793, 14.816]
  MoveL 560 to (721.09, 228.01, 0) mm, rotated rx 0 ry 90 rz -60.43 deg; joints [28.442, -49.147, 112.744, -34.887, -67.842, 14.734]
  MoveL 561 to (718.54, 227.44, 0) mm, rotated rx 0 ry 90 rz -60.43 deg; joints [28.512, -49.228, 112.916, -34.793, -67.899, 14.651]
  MoveL 562 to (715.95, 227.1, 0) mm, rotated rx 0 ry 90 rz -60.43 deg; joints [28.575, -49.314, 113.1, -34.705, -67.963, 14.566]
  MoveL 563 to (444.31, 344.54, 0) mm, rotated rx 0 ry 90 rz -60.43 deg; joints [29.968, -60.204, 136.911, -31.145, -78.569, 6.83]
  Set speed (60.0 mm/s)
  MoveL 564 to (442.29, 347.38, 0) mm, rotated rx 0 ry 90 rz -60.43 deg; joints [29.892, -60.31, 137.152, -31.207, -78.693, 6.773]
  MoveL 565 to (440.09, 350.06, 0) mm, rotated rx 0 ry 90 rz -60.43 deg; joints [29.828, -60.418, 137.399, -31.258, -78.819, 6.713]
  MoveL 566 to (435.19, 354.95, 0) mm, rotated rx 0 ry 90 rz -60.43 deg; joints [29.733, -60.639, 137.906, -31.325, -79.075, 6.58]
  MoveL 567 to (429.7, 359.17, 0) mm, rotated rx 0 ry 90 rz -60.43 deg; joints [29.683, -60.865, 138.425, -31.346, -79.331, 6.434]
  MoveL 568 to (423.7, 362.68, 0) mm, rotated rx 0 ry 90 rz -60.43 deg; joints [29.679, -61.093, 138.95, -31.322, -79.585, 6.278]
  MoveL 569 to (417.35, 365.42, 0) mm, rotated rx 0 ry 90 rz -60.43 deg; joints [29.72, -61.317, 139.468, -31.253, -79.832, 6.115]
  MoveL 570 to (410.73, 367.39, 0) mm, rotated rx 0 ry 90 rz -60.43 deg; joints [29.805, -61.535, 139.974, -31.141, -80.069, 5.949]
  MoveL 571 to (403.93, 368.58, 0) mm, rotated rx 0 ry 90 rz -60.43 deg; joints [29.932, -61.745, 140.461, -30.987, -80.294, 5.782]
  MoveL 572 to (397.02, 368.98, 0) mm, rotated rx 0 ry 90 rz -60.43 deg; joints [30.102, -61.943, 140.924, -30.793, -80.504, 5.616]
  MoveL 573 to (223.67, 368.98, 0) mm, rotated rx 0 ry 90 rz -60.43 deg; joints [35.626, -66.306, 151.62, -24.875, -85.746, 1.97]
  MoveL 574 to (223.67, 407.08, 0) mm, rotated rx 0 ry 90 rz -60.43 deg; joints [33.613, -66.894, 153.176, -26.864, -86.682, 1.679]
  MoveL 575 to (451.51, 407.08, 0) mm, rotated rx 0 ry 90 rz -60.43 deg; joints [26.897, -60.98, 138.69, -34.145, -79.779, 6.862]
  MoveL 576 to (619.38, 153.08, 0) mm, rotated rx 0 ry 90 rz -60.43 deg; joints [33.294, -51.118, 116.947, -29.325, -68.629, 11.568]
  MoveL 577 to (570.85, 153.08, 0) mm, rotated rx 0 ry 90 rz -60.43 deg; joints [34.458, -52.692, 120.325, -27.777, -69.995, 10.215]
  MoveL 578 to (444.31, 344.54, 0) mm, rotated rx 0 ry 90 rz -60.43 deg; joints [29.968, -60.204, 136.911, -31.145, -78.569, 6.83]
  MoveL 579 to (791.94, 89.58, 0) mm, rotated rx 0 ry 90 rz -60.43 deg; joints [31.735, -43.492, 100.829, -33.03, -61.743, 17.108]
  Set speed (60.0 mm/s)
  MoveL 580 to (791.94, 127.68, 0) mm, rotated rx 0 ry 90 rz -60.43 deg; joints [30.507, -44.384, 102.697, -34.072, -62.918, 17.114]
  MoveL 581 to (569.33, 127.68, 0) mm, rotated rx 0 ry 90 rz -60.43 deg; joints [35.401, -52.177, 119.218, -26.888, -69.302, 10.161]
  MoveL 582 to (555.62, 129.27, 0) mm, rotated rx 0 ry 90 rz -60.43 deg; joints [35.691, -52.644, 120.224, -26.492, -69.732, 9.796]
  MoveL 583 to (549, 131.24, 0) mm, rotated rx 0 ry 90 rz -60.43 deg; joints [35.791, -52.895, 120.765, -26.341, -69.975, 9.622]
  MoveL 584 to (542.65, 133.98, 0) mm, rotated rx 0 ry 90 rz -60.43 deg; joints [35.856, -53.154, 121.323, -26.224, -70.233, 9.458]
  MoveL 585 to (536.65, 137.49, 0) mm, rotated rx 0 ry 90 rz -60.43 deg; joints [35.886, -53.417, 121.892, -26.145, -70.503, 9.304]
  MoveL 586 to (531.16, 141.71, 0) mm, rotated rx 0 ry 90 rz -60.43 deg; joints [35.877, -53.68, 122.46, -26.107, -70.779, 9.165]
  MoveL 587 to (526.26, 146.6, 0) mm, rotated rx 0 ry 90 rz -60.43 deg; joints [35.828, -53.938, 123.019, -26.112, -71.057, 9.041]
  MoveL 588 to (522.04, 152.12, 0) mm, rotated rx 0 ry 90 rz -60.43 deg; joints [35.737, -54.188, 123.561, -26.162, -71.333, 8.936]
  MoveL 589 to (395.5, 343.58, 0) mm, rotated rx 0 ry 90 rz -60.43 deg; joints [31.33, -61.567, 140.049, -29.596, -79.951, 5.66]
  MoveL 590 to (346.97, 343.58, 0) mm, rotated rx 0 ry 90 rz -60.43 deg; joints [32.749, -62.875, 143.12, -28.025, -81.37, 4.566]
  MoveL 591 to (514.85, 89.58, 0) mm, rotated rx 0 ry 90 rz -60.43 deg; joints [38.154, -52.981, 120.949, -23.84, -69.688, 8.72]
  MoveL 592 to (791.94, 89.58, 0) mm, rotated rx 0 ry 90 rz -60.43 deg; joints [31.735, -43.492, 100.829, -33.03, -61.743, 17.108]
  MoveL 593 to (893.34, 291.99, 0) mm, rotated rx 0 ry 90 rz -60.43 deg; joints [23.248, -43.651, 101.163, -41.963, -64.663, 21.048]
  Set speed (60.0 mm/s)
  MoveL 594 to (890.74, 291.64, 0) mm, rotated rx 0 ry 90 rz -60.43 deg; joints [23.298, -43.754, 101.377, -41.875, -64.728, 20.943]
  MoveL 595 to (888.19, 291.08, 0) mm, rotated rx 0 ry 90 rz -60.43 deg; joints [23.356, -43.85, 101.579, -41.783, -64.786, 20.84]
  MoveL 596 to (885.71, 290.29, 0) mm, rotated rx 0 ry 90 rz -60.43 deg; joints [23.42, -43.939, 101.766, -41.686, -64.836, 20.74]
  MoveL 597 to (883.3, 289.29, 0) mm, rotated rx 0 ry 90 rz -60.43 deg; joints [23.491, -44.021, 101.937, -41.585, -64.878, 20.643]
  MoveL 598 to (881, 288.07, 0) mm, rotated rx 0 ry 90 rz -60.43 deg; joints [23.568, -44.095, 102.091, -41.48, -64.911, 20.551]
  MoveL 599 to (878.81, 286.63, 0) mm, rotated rx 0 ry 90 rz -60.43 deg; joints [23.651, -44.159, 102.226, -41.373, -64.935, 20.463]
  MoveL 600 to (876.76, 284.98, 0) mm, rotated rx 0 ry 90 rz -60.43 deg; joints [23.739, -44.214, 102.341, -41.263, -64.949, 20.38]
  MoveL 601 to (874.88, 283.15, 0) mm, rotated rx 0 ry 90 rz -60.43 deg; joints [23.831, -44.258, 102.433, -41.153, -64.953, 20.305]
  MoveL 602 to (873.22, 281.16, 0) mm, rotated rx 0 ry 90 rz -60.43 deg; joints [23.925, -44.29, 102.501, -41.044, -64.947, 20.238]
  MoveL 603 to (871.77, 279.02, 0) mm, rotated rx 0 ry 90 rz -60.43 deg; joints [24.022, -44.311, 102.544, -40.938, -64.931, 20.179]
  MoveL 604 to (870.55, 276.75, 0) mm, rotated rx 0 ry 90 rz -60.43 deg; joints [24.119, -44.319, 102.561, -40.834, -64.904, 20.13]
  MoveL 605 to (869.59, 274.37, 0) mm, rotated rx 0 ry 90 rz -60.43 deg; joints [24.216, -44.315, 102.552, -40.735, -64.867, 20.091]
  MoveL 606 to (868.88, 271.89, 0) mm, rotated rx 0 ry 90 rz -60.43 deg; joints [24.313, -44.298, 102.517, -40.64, -64.82, 20.061]
  MoveL 607 to (868.44, 269.33, 0) mm, rotated rx 0 ry 90 rz -60.43 deg; joints [24.408, -44.268, 102.455, -40.551, -64.763, 20.043]
  MoveL 608 to (868.3, 266.7, 0) mm, rotated rx 0 ry 90 rz -60.43 deg; joints [24.501, -44.225, 102.365, -40.469, -64.695, 20.035]
  MoveL 609 to (868.3, 25.4, 0) mm, rotated rx 0 ry 90 rz -60.43 deg; joints [32.242, -38.75, 90.953, -34.144, -57.304, 20.12]
  MoveL 610 to (817.34, 25.4, 0) mm, rotated rx 0 ry 90 rz -60.43 deg; joints [33.224, -40.867, 95.353, -32.273, -58.892, 18.07]
  MoveL 611 to (817.34, 330.2, 0) mm, rotated rx 0 ry 90 rz -60.43 deg; joints [23.045, -47.38, 109.002, -40.973, -67.811, 18.159]
  MoveL 612 to (983.12, 330.2, 0) mm, rotated rx 0 ry 90 rz -60.43 deg; joints [20.716, -40.403, 94.386, -45.76, -63.106, 24.915]
  MoveL 613 to (1117.42, 127, 0) mm, rotated rx 0 ry 90 rz -60.43 deg; joints [25.259, -29.069, 70.997, -46.521, -52.543, 32.674]
  MoveL 614 to (1068.89, 127, 0) mm, rotated rx 0 ry 90 rz -60.43 deg; joints [25.934, -31.816, 76.638, -44.268, -54.226, 29.677]
  MoveL 615 to (967.85, 279.88, 0) mm, rotated rx 0 ry 90 rz -60.43 deg; joints [22.594, -40.189, 93.942, -43.921, -62.162, 24.214]
  MoveL 616 to (965.72, 282.67, 0) mm, rotated rx 0 ry 90 rz -60.43 deg; joints [22.531, -40.337, 94.25, -43.927, -62.303, 24.118]
  MoveL 617 to (963.26, 285.11, 0) mm, rotated rx 0 ry 90 rz -60.43 deg; joints [22.484, -40.494, 94.575, -43.915, -62.444, 24.009]
  MoveL 618 to (960.53, 287.21, 0) mm, rotated rx 0 ry 90 rz -60.43 deg; joints [22.451, -40.655, 94.912, -43.885, -62.583, 23.888]
  MoveL 619 to (957.55, 288.94, 0) mm, rotated rx 0 ry 90 rz -60.43 deg; joints [22.435, -40.82, 95.255, -43.838, -62.718, 23.756]
  MoveL 620 to (954.39, 290.31, 0) mm, rotated rx 0 ry 90 rz -60.43 deg; joints [22.433, -40.987, 95.601, -43.776, -62.849, 23.618]
  MoveL 621 to (951.08, 291.3, 0) mm, rotated rx 0 ry 90 rz -60.43 deg; joints [22.445, -41.152, 95.945, -43.7, -62.973, 23.473]
  MoveL 622 to (947.67, 291.9, 0) mm, rotated rx 0 ry 90 rz -60.43 deg; joints [22.472, -41.314, 96.282, -43.61, -63.089, 23.324]
  MoveL 623 to (944.2, 292.1, 0) mm, rotated rx 0 ry 90 rz -60.43 deg; joints [22.514, -41.47, 96.609, -43.508, -63.195, 23.174]
  MoveL 624 to (895.95, 292.1, 0) mm, rotated rx 0 ry 90 rz -60.43 deg; joints [23.206, -43.544, 100.938, -42.044, -64.59, 21.154]
  MoveL 625 to (893.34, 291.99, 0) mm, rotated rx 0 ry 90 rz -60.43 deg; joints [23.248, -43.651, 101.163, -41.963, -64.663, 21.048]
  MoveL 626 to (1117.81, 63.61, 0) mm, rotated rx 0 ry 90 rz -60.43 deg; joints [27.05, -27.16, 67.085, -45.751, -50.179, 33.321]
  Set speed (60.0 mm/s)
  MoveL 627 to (1115.19, 63.5, 0) mm, rotated rx 0 ry 90 rz -60.43 deg; joints [27.091, -27.318, 67.409, -45.608, -50.272, 33.138]
  MoveL 628 to (1066.94, 63.5, 0) mm, rotated rx 0 ry 90 rz -60.43 deg; joints [27.797, -30.151, 73.217, -43.159, -52.03, 29.982]
  MoveL 629 to (1060.06, 64.3, 0) mm, rotated rx 0 ry 90 rz -60.43 deg; joints [27.878, -30.557, 74.051, -42.843, -52.303, 29.558]
  MoveL 630 to (1056.75, 65.29, 0) mm, rotated rx 0 ry 90 rz -60.43 deg; joints [27.899, -30.768, 74.485, -42.703, -52.455, 29.352]
  MoveL 631 to (1053.59, 66.65, 0) mm, rotated rx 0 ry 90 rz -60.43 deg; joints [27.908, -30.981, 74.922, -42.577, -52.616, 29.155]
  MoveL 632 to (1050.62, 68.39, 0) mm, rotated rx 0 ry 90 rz -60.43 deg; joints [27.904, -31.193, 75.357, -42.467, -52.783, 28.968]
  MoveL 633 to (1047.88, 70.49, 0) mm, rotated rx 0 ry 90 rz -60.43 deg; joints [27.885, -31.401, 75.785, -42.375, -52.954, 28.795]
  MoveL 634 to (1045.42, 72.93, 0) mm, rotated rx 0 ry 90 rz -60.43 deg; joints [27.852, -31.603, 76.199, -42.303, -53.127, 28.637]
  MoveL 635 to (1043.29, 75.72, 0) mm, rotated rx 0 ry 90 rz -60.43 deg; joints [27.804, -31.795, 76.595, -42.254, -53.301, 28.498]
  MoveL 636 to (942.25, 228.6, 0) mm, rotated rx 0 ry 90 rz -60.43 deg; joints [24.644, -40.331, 94.237, -41.734, -61.452, 23.089]
  MoveL 637 to (893.72, 228.6, 0) mm, rotated rx 0 ry 90 rz -60.43 deg; joints [25.39, -42.431, 98.612, -40.165, -62.89, 21.038]
  MoveL 638 to (1028.02, 25.4, 0) mm, rotated rx 0 ry 90 rz -60.43 deg; joints [29.478, -31.143, 75.254, -40.746, -51.993, 27.946]
  MoveL 639 to (1193.8, 25.4, 0) mm, rotated rx 0 ry 90 rz -60.43 deg; joints [27.035, -20.475, 53.43, -50.471, -45.527, 40.331]
  MoveL 640 to (1193.8, 330.2, 0) mm, rotated rx 0 ry 90 rz -60.43 deg; joints [18.337, -29.365, 71.604, -53.344, -56.675, 36.437]
  MoveL 641 to (1142.85, 330.2, 0) mm, rotated rx 0 ry 90 rz -60.43 deg; joints [18.863, -32.359, 77.754, -51.24, -58.306, 33.2]
  MoveL 642 to (1142.85, 88.9, 0) mm, rotated rx 0 ry 90 rz -60.43 deg; joints [25.994, -26.376, 65.48, -47.387, -50.206, 34.827]
  MoveL 643 to (1142.7, 86.27, 0) mm, rotated rx 0 ry 90 rz -60.43 deg; joints [26.07, -26.303, 65.33, -47.353, -50.111, 34.848]
  MoveL 644 to (1142.26, 83.71, 0) mm, rotated rx 0 ry 90 rz -60.43 deg; joints [26.147, -26.25, 65.222, -47.304, -50.029, 34.848]
  MoveL 645 to (1141.56, 81.23, 0) mm, rotated rx 0 ry 90 rz -60.43 deg; joints [26.226, -26.217, 65.154, -47.241, -49.961, 34.827]
  MoveL 646 to (1140.59, 78.85, 0) mm, rotated rx 0 ry 90 rz -60.43 deg; joints [26.306, -26.203, 65.127, -47.164, -49.906, 34.785]
  MoveL 647 to (1139.37, 76.58, 0) mm, rotated rx 0 ry 90 rz -60.43 deg; joints [26.386, -26.209, 65.139, -47.074, -49.864, 34.724]
  MoveL 648 to (1137.93, 74.44, 0) mm, rotated rx 0 ry 90 rz -60.43 deg; joints [26.466, -26.234, 65.19, -46.972, -49.837, 34.644]
  MoveL 649 to (1136.26, 72.45, 0) mm, rotated rx 0 ry 90 rz -60.43 deg; joints [26.544, -26.277, 65.278, -46.86, -49.823, 34.546]
  MoveL 650 to (1134.38, 70.61, 0) mm, rotated rx 0 ry 90 rz -60.43 deg; joints [26.621, -26.339, 65.404, -46.737, -49.823, 34.431]
  MoveL 651 to (1132.33, 68.97, 0) mm, rotated rx 0 ry 90 rz -60.43 deg; joints [26.696, -26.417, 65.564, -46.606, -49.837, 34.301]
  MoveL 652 to (1130.15, 67.53, 0) mm, rotated rx 0 ry 90 rz -60.43 deg; joints [26.766, -26.51, 65.755, -46.47, -49.865, 34.159]
  MoveL 653 to (1127.84, 66.31, 0) mm, rotated rx 0 ry 90 rz -60.43 deg; joints [26.833, -26.617, 65.974, -46.33, -49.905, 34.006]
  MoveL 654 to (1125.43, 65.31, 0) mm, rotated rx 0 ry 90 rz -60.43 deg; joints [26.895, -26.737, 66.219, -46.186, -49.957, 33.845]
  MoveL 655 to (1122.95, 64.52, 0) mm, rotated rx 0 ry 90 rz -60.43 deg; joints [26.952, -26.868, 66.488, -46.041, -50.02, 33.676]
  MoveL 656 to (1120.4, 63.96, 0) mm, rotated rx 0 ry 90 rz -60.43 deg; joints [27.004, -27.01, 66.777, -45.896, -50.095, 33.501]
  MoveL 657 to (1117.81, 63.61, 0) mm, rotated rx 0 ry 90 rz -60.43 deg; joints [27.05, -27.16, 67.085, -45.751, -50.179, 33.321]
  MoveL 658 to (774.66, 25.4, 0) mm, rotated rx 0 ry 90 rz -60.43 deg; joints [34.087, -42.552, 98.864, -30.755, -60.194, 16.477]
  Set speed (60.0 mm/s)
  MoveL 659 to (464.73, 25.4, 0) mm, rotated rx 0 ry 90 rz -60.43 deg; joints [41.727, -52.874, 120.72, -20.077, -69.072, 7.438]
  MoveL 660 to (296.85, 279.4, 0) mm, rotated rx 0 ry 90 rz -60.43 deg; joints [37.33, -63.006, 143.431, -23.39, -81.199, 3.786]
  MoveL 661 to (345.39, 279.4, 0) mm, rotated rx 0 ry 90 rz -60.43 deg; joints [35.73, -61.772, 140.524, -25.123, -79.793, 4.75]
  MoveL 662 to (471.92, 87.94, 0) mm, rotated rx 0 ry 90 rz -60.43 deg; joints [39.407, -54.21, 123.609, -22.32, -70.826, 7.679]
  MoveL 663 to (476.14, 82.42, 0) mm, rotated rx 0 ry 90 rz -60.43 deg; joints [39.478, -53.956, 123.058, -22.285, -70.542, 7.774]
  MoveL 664 to (481.04, 77.53, 0) mm, rotated rx 0 ry 90 rz -60.43 deg; joints [39.508, -53.696, 122.494, -22.295, -70.257, 7.886]
  MoveL 665 to (486.53, 73.31, 0) mm, rotated rx 0 ry 90 rz -60.43 deg; joints [39.497, -53.433, 121.927, -22.348, -69.976, 8.013]
  MoveL 666 to (492.53, 69.8, 0) mm, rotated rx 0 ry 90 rz -60.43 deg; joints [39.448, -53.172, 121.362, -22.442, -69.702, 8.154]
  MoveL 667 to (498.88, 67.06, 0) mm, rotated rx 0 ry 90 rz -60.43 deg; joints [39.364, -52.918, 120.813, -22.573, -69.442, 8.305]
  MoveL 668 to (505.5, 65.09, 0) mm, rotated rx 0 ry 90 rz -60.43 deg; joints [39.247, -52.673, 120.285, -22.738, -69.198, 8.465]
  MoveL 669 to (519.21, 63.5, 0) mm, rotated rx 0 ry 90 rz -60.43 deg; joints [38.925, -52.223, 119.316, -23.157, -68.768, 8.805]
  MoveL 670 to (774.66, 63.5, 0) mm, rotated rx 0 ry 90 rz -60.43 deg; joints [32.906, -43.522, 100.892, -31.746, -61.433, 16.482]
  MoveL 671 to (774.66, 25.4, 0) mm, rotated rx 0 ry 90 rz -60.43 deg; joints [34.087, -42.552, 98.864, -30.755, -60.194, 16.477]
  Set speed (2000.0 mm/s)
  MoveL 672 to (774.66, 25.4, 0) mm, rotated rx 0 ry 90 rz -60.43 deg; joints [34.087, -42.552, 98.864, -30.755, -60.194, 16.477]
  MoveL 673 to (774.66, 25.4, 10) mm, rotated rx 0 ry 90 rz -60.43 deg; joints [34.087, -43.037, 98.882, -30.893, -59.792, 16.754]
